LIN {X 0,Y 572.923,Z 346.522,A -85,B 0,C 180,E1 -2106.073,E2 -2106.073} C_VEL
LIN {X 0,Y 572.929,Z 346.988,A -85,B 0,C 180,E1 -2107.123,E2 -2107.123} C_VEL
LIN {X 0,Y 572.933,Z 346.186,A -85,B 0,C 180,E1 -2108.272,E2 -2108.272} C_VEL
LIN {X 0,Y 572.946,Z 344.14,A -85,B 0,C 180,E1 -2109.395,E2 -2109.395} C_VEL
LIN {X 0,Y 573.006,Z 340.639,A -85,B 0,C 180,E1 -2110.546,E2 -2110.546} C_VEL
LIN {X 0,Y 573.022,Z 335.263,A -85,B 0,C 180,E1 -2111.743,E2 -2111.743} C_VEL
LIN {X 0,Y 573.058,Z 329.01,A -85,B 0,C 180,E1 -2112.77,E2 -2112.77} C_VEL
LIN {X 0,Y 573.128,Z 322.073,A -85,B 0,C 180,E1 -2113.656,E2 -2113.656} C_VEL
LIN {X 0,Y 573.173,Z 315.507,A -85,B 0,C 180,E1 -2114.34,E2 -2114.34} C_VEL
LIN {X 0,Y 573.239,Z 307.033,A -85,B 0,C 180,E1 -2115.058,E2 -2115.058} C_VEL
LIN {X 0,Y 573.328,Z 297.887,A -85,B 0,C 180,E1 -2115.675,E2 -2115.675} C_VEL
LIN {X 0,Y 573.423,Z 286.508,A -85,B 0,C 180,E1 -2116.263,E2 -2116.263} C_VEL
LIN {X 0,Y 573.486,Z 274.83,A -85,B 0,C 180,E1 -2116.68,E2 -2116.68} C_VEL
LIN {X 0,Y 573.2,Z 269.025,A -85,B 0,C 180,E1 -2116.842,E2 -2116.842} C_VEL
LIN {X 0,Y 573.003,Z 267.326,A -85,B 0,C 180,E1 -2116.901,E2 -2116.901} C_VEL
LIN {X 0,Y 572.997,Z 260.215,A -85,B 0,C 180,E1 -2119.939,E2 -2119.939} C_VEL
LIN {X 0,Y 572.989,Z 255.042,A -85,B 0,C 180,E1 -2122.173,E2 -2122.173} C_VEL
LIN {X 0,Y 573.027,Z 247.981,A -85,B 0,C 180,E1 -2125.259,E2 -2125.259} C_VEL
LIN {X 0,Y 573.063,Z 241.461,A -85,B 0,C 180,E1 -2128.173,E2 -2128.173} C_VEL
LIN {X 0,Y 573.075,Z 235.778,A -85,B 0,C 180,E1 -2130.623,E2 -2130.623} C_VEL
LIN {X 0,Y 573.068,Z 230.379,A -85,B 0,C 180,E1 -2133.014,E2 -2133.014} C_VEL
LIN {X 0,Y 573.079,Z 224.661,A -85,B 0,C 180,E1 -2135.357,E2 -2135.357} C_VEL
LIN {X 0,Y 573.108,Z 218.041,A -85,B 0,C 180,E1 -2138.036,E2 -2138.036} C_VEL
LIN {X 0,Y 573.12,Z 217.1,A -85,B 0,C 180,E1 -2138.415,E2 -2138.415} C_VEL
LIN {X 0,Y 573.273,Z 217.077,A -85,B 0,C 180,E1 -2140.731,E2 -2140.731} C_VEL
LIN {X 0,Y 573.248,Z 217.082,A -85,B 0,C 180,E1 -2143.621,E2 -2143.621} C_VEL
LIN {X 0,Y 573.231,Z 217.082,A -85,B 0,C 180,E1 -2146.529,E2 -2146.529} C_VEL
LIN {X 0,Y 573.267,Z 217.078,A -85,B 0,C 180,E1 -2148.745,E2 -2148.745} C_VEL
LIN {X 0,Y 573.286,Z 217.076,A -85,B 0,C 180,E1 -2151.54,E2 -2151.54} C_VEL
LIN {X 0,Y 573.284,Z 217.077,A -85,B 0,C 180,E1 -2154.372,E2 -2154.372} C_VEL
LIN {X 0,Y 573.315,Z 217.073,A -85,B 0,C 180,E1 -2157.892,E2 -2157.892} C_VEL
LIN {X 0,Y 573.327,Z 217.07,A -85,B 0,C 180,E1 -2160.702,E2 -2160.702} C_VEL
LIN {X 0,Y 573.307,Z 217.073,A -85,B 0,C 180,E1 -2162.811,E2 -2162.811} C_VEL
LIN {X 0,Y 573.288,Z 217.075,A -85,B 0,C 180,E1 -2165.628,E2 -2165.628} C_VEL
LIN {X 0,Y 573.286,Z 217.078,A -85,B 0,C 180,E1 -2168.459,E2 -2168.459} C_VEL
LIN {X 0,Y 573.276,Z 217.076,A -85,B 0,C 180,E1 -2171.312,E2 -2171.312} C_VEL
LIN {X 0,Y 573.286,Z 217.078,A -85,B 0,C 180,E1 -2174.424,E2 -2174.424} C_VEL
LIN {X 0,Y 573.262,Z 217.079,A -85,B 0,C 180,E1 -2177.111,E2 -2177.111} C_VEL
LIN {X 0,Y 573.246,Z 217.081,A -85,B 0,C 180,E1 -2180.077,E2 -2180.077} C_VEL
LIN {X 0,Y 573.237,Z 217.081,A -85,B 0,C 180,E1 -2182.338,E2 -2182.338} C_VEL
LIN {X 0,Y 573.244,Z 217.081,A -85,B 0,C 180,E1 -2185.411,E2 -2185.411} C_VEL
LIN {X 0,Y 573.239,Z 217.084,A -85,B 0,C 180,E1 -2188.564,E2 -2188.564} C_VEL
LIN {X 0,Y 573.223,Z 217.086,A -85,B 0,C 180,E1 -2190.994,E2 -2190.994} C_VEL
LIN {X 0,Y 573.243,Z 217.083,A -85,B 0,C 180,E1 -2193.521,E2 -2193.521} C_VEL
LIN {X 0,Y 573.218,Z 217.084,A -85,B 0,C 180,E1 -2196.051,E2 -2196.051} C_VEL
LIN {X 0,Y 573.246,Z 217.08,A -85,B 0,C 180,E1 -2198.701,E2 -2198.701} C_VEL
LIN {X 0,Y 573.231,Z 217.084,A -85,B 0,C 180,E1 -2201.593,E2 -2201.593} C_VEL
LIN {X 0,Y 573.236,Z 217.083,A -85,B 0,C 180,E1 -2204.334,E2 -2204.334} C_VEL
LIN {X 0,Y 573.244,Z 217.081,A -85,B 0,C 180,E1 -2207.358,E2 -2207.358} C_VEL
LIN {X 0,Y 573.253,Z 217.079,A -85,B 0,C 180,E1 -2210.568,E2 -2210.568} C_VEL
LIN {X 0,Y 573.279,Z 217.182,A -85,B 0,C 180,E1 -2213.244,E2 -2213.244} C_VEL
LIN {X 0,Y 573.748,Z 221.859,A -85,B 0,C 180,E1 -2214.85,E2 -2214.85} C_VEL
LIN {X 0,Y 573.7,Z 228.345,A -85,B 0,C 180,E1 -2216.966,E2 -2216.966} C_VEL
LIN {X 0,Y 573.556,Z 237.515,A -85,B 0,C 180,E1 -2219.842,E2 -2219.842} C_VEL
LIN {X 0,Y 573.422,Z 246.743,A -85,B 0,C 180,E1 -2222.638,E2 -2222.638} C_VEL
LIN {X 0,Y 573.367,Z 256.185,A -85,B 0,C 180,E1 -2225.37,E2 -2225.37} C_VEL
LIN {X 0,Y 573.349,Z 265.605,A -85,B 0,C 180,E1 -2228.046,E2 -2228.046} C_VEL
LIN {X 0,Y 573.228,Z 276.33,A -85,B 0,C 180,E1 -2231.078,E2 -2231.078} C_VEL
LIN {X 0,Y 573.164,Z 286.788,A -85,B 0,C 180,E1 -2233.985,E2 -2233.985} C_VEL
LIN {X 0,Y 573.094,Z 297.379,A -85,B 0,C 180,E1 -2236.887,E2 -2236.887} C_VEL
LIN {X 0,Y 573.083,Z 299.53,A -85,B 0,C 180,E1 -2237.472,E2 -2237.472} C_VEL
LIN {X 0,Y 573.866,Z 306.371,A -85,B 0,C 180,E1 -2237.624,E2 -2237.624} C_VEL
LIN {X 0,Y 573.779,Z 318.5,A -85,B 0,C 180,E1 -2237.937,E2 -2237.937} C_VEL
LIN {X 0,Y 573.642,Z 330.524,A -85,B 0,C 180,E1 -2238.382,E2 -2238.382} C_VEL
LIN {X 0,Y 573.509,Z 342.485,A -85,B 0,C 180,E1 -2238.977,E2 -2238.977} C_VEL
LIN {X 0,Y 573.446,Z 353.483,A -85,B 0,C 180,E1 -2239.675,E2 -2239.675} C_VEL
LIN {X 0,Y 573.308,Z 363.647,A -85,B 0,C 180,E1 -2240.474,E2 -2240.474} C_VEL
LIN {X 0,Y 573.215,Z 372.787,A -85,B 0,C 180,E1 -2241.362,E2 -2241.362} C_VEL
LIN {X 0,Y 573.142,Z 381.69,A -85,B 0,C 180,E1 -2242.425,E2 -2242.425} C_VEL
LIN {X 0,Y 573.051,Z 388.404,A -85,B 0,C 180,E1 -2243.415,E2 -2243.415} C_VEL
LIN {X 0,Y 573.07,Z 393.68,A -85,B 0,C 180,E1 -2244.37,E2 -2244.37} C_VEL
LIN {X 0,Y 573.028,Z 398.372,A -85,B 0,C 180,E1 -2245.428,E2 -2245.428} C_VEL
LIN {X 0,Y 573.022,Z 401.958,A -85,B 0,C 180,E1 -2246.484,E2 -2246.484} C_VEL
LIN {X 0,Y 572.959,Z 403.808,A -85,B 0,C 180,E1 -2247.188,E2 -2247.188} C_VEL
LIN {X 0,Y 572.94,Z 405.198,A -85,B 0,C 180,E1 -2247.891,E2 -2247.891} C_VEL
LIN {X 0,Y 572.94,Z 406.785,A -85,B 0,C 180,E1 -2249.297,E2 -2249.297} C_VEL
LIN {X 0,Y 572.938,Z 407,A -85,B 0,C 180,E1 -2250,E2 -2250} C_VEL
LIN {X 0,Y 572.946,Z 406.186,A -85,B 0,C 180,E1 -2251.406,E2 -2251.406} C_VEL
LIN {X 0,Y 572.94,Z 405.199,A -85,B 0,C 180,E1 -2252.109,E2 -2252.109} C_VEL
LIN {X 0,Y 572.959,Z 403.81,A -85,B 0,C 180,E1 -2252.812,E2 -2252.812} C_VEL
LIN {X 0,Y 573.015,Z 400.895,A -85,B 0,C 180,E1 -2253.868,E2 -2253.868} C_VEL
LIN {X 0,Y 572.963,Z 396.948,A -85,B 0,C 180,E1 -2254.926,E2 -2254.926} C_VEL
LIN {X 0,Y 573.065,Z 390.876,A -85,B 0,C 180,E1 -2256.16,E2 -2256.16} C_VEL
LIN {X 0,Y 573.119,Z 384.236,A -85,B 0,C 180,E1 -2257.221,E2 -2257.221} C_VEL
LIN {X 0,Y 573.201,Z 375.989,A -85,B 0,C 180,E1 -2258.283,E2 -2258.283} C_VEL
LIN {X 0,Y 573.287,Z 367.537,A -85,B 0,C 180,E1 -2259.17,E2 -2259.17} C_VEL
LIN {X 0,Y 573.425,Z 357.096,A -85,B 0,C 180,E1 -2260.058,E2 -2260.058} C_VEL
LIN {X 0,Y 573.511,Z 345.53,A -85,B 0,C 180,E1 -2260.847,E2 -2260.847} C_VEL
LIN {X 0,Y 573.61,Z 333.88,A -85,B 0,C 180,E1 -2261.466,E2 -2261.466} C_VEL
LIN {X 0,Y 573.758,Z 321.166,A -85,B 0,C 180,E1 -2261.974,E2 -2261.974} C_VEL
LIN {X 0,Y 573.867,Z 308.51,A -85,B 0,C 180,E1 -2262.331,E2 -2262.331} C_VEL
LIN {X 0,Y 573.573,Z 302.638,A -85,B 0,C 180,E1 -2262.455,E2 -2262.455} C_VEL
LIN {X 0,Y 573.084,Z 299.529,A -85,B 0,C 180,E1 -2262.528,E2 -2262.528} C_VEL
LIN {X 0,Y 573.158,Z 289.435,A -85,B 0,C 180,E1 -2265.286,E2 -2265.286} C_VEL
LIN {X 0,Y 573.217,Z 278.843,A -85,B 0,C 180,E1 -2268.219,E2 -2268.219} C_VEL
LIN {X 0,Y 573.3,Z 269.576,A -85,B 0,C 180,E1 -2270.825,E2 -2270.825} C_VEL
LIN {X 0,Y 573.349,Z 260.089,A -85,B 0,C 180,E1 -2273.477,E2 -2273.477} C_VEL
LIN {X 0,Y 573.356,Z 249.227,A -85,B 0,C 180,E1 -2276.516,E2 -2276.516} C_VEL
LIN {X 0,Y 573.441,Z 239.004,A -85,B 0,C 180,E1 -2279.522,E2 -2279.522} C_VEL
LIN {X 0,Y 573.633,Z 230.314,A -85,B 0,C 180,E1 -2282.288,E2 -2282.288} C_VEL
LIN {X 0,Y 573.793,Z 223.076,A -85,B 0,C 180,E1 -2284.851,E2 -2284.851} C_VEL
LIN {X 0,Y 573.73,Z 220.074,A -85,B 0,C 180,E1 -2286.052,E2 -2286.052} C_VEL
LIN {X 0,Y 573.256,Z 217.082,A -85,B 0,C 180,E1 -2287.457,E2 -2287.457} C_VEL
LIN {X 0,Y 573.248,Z 217.083,A -85,B 0,C 180,E1 -2290.525,E2 -2290.525} C_VEL
LIN {X 0,Y 573.242,Z 217.082,A -85,B 0,C 180,E1 -2293.359,E2 -2293.359} C_VEL
LIN {X 0,Y 573.243,Z 217.081,A -85,B 0,C 180,E1 -2296.332,E2 -2296.332} C_VEL
LIN {X 0,Y 573.233,Z 217.082,A -85,B 0,C 180,E1 -2298.543,E2 -2298.543} C_VEL
LIN {X 0,Y 573.247,Z 217.081,A -85,B 0,C 180,E1 -2301.299,E2 -2301.299} C_VEL
LIN {X 0,Y 573.217,Z 217.086,A -85,B 0,C 180,E1 -2304.019,E2 -2304.019} C_VEL
LIN {X 0,Y 573.17,Z 217.102,A -85,B 0,C 180,E1 -2305.665,E2 -2305.665} C_VEL
LIN {X 0,Y 573.151,Z 219.81,A -85,B 0,C 180,E1 -2308.179,E2 -2308.179} C_VEL
LIN {X 0,Y 573.114,Z 222.452,A -85,B 0,C 180,E1 -2310.626,E2 -2310.626} C_VEL
LIN {X 0,Y 573.064,Z 225.599,A -85,B 0,C 180,E1 -2313.543,E2 -2313.543} C_VEL
LIN {X 0,Y 573.028,Z 228.468,A -85,B 0,C 180,E1 -2316.126,E2 -2316.126} C_VEL
LIN {X 0,Y 572.987,Z 231.649,A -85,B 0,C 180,E1 -2319.164,E2 -2319.164} C_VEL
LIN {X 0,Y 572.947,Z 234.241,A -85,B 0,C 180,E1 -2321.402,E2 -2321.402} C_VEL
LIN {X 0,Y 572.957,Z 237.107,A -85,B 0,C 180,E1 -2323.613,E2 -2323.613} C_VEL
LIN {X 0,Y 572.983,Z 240.932,A -85,B 0,C 180,E1 -2326.523,E2 -2326.523} C_VEL
LIN {X 0,Y 572.961,Z 243.669,A -85,B 0,C 180,E1 -2328.581,E2 -2328.581} C_VEL
LIN {X 0,Y 573.844,Z 250.337,A -85,B 0,C 180,E1 -2328.759,E2 -2328.759} C_VEL
LIN {X 0,Y 573.776,Z 263.544,A -85,B 0,C 180,E1 -2329.153,E2 -2329.153} C_VEL
LIN {X 0,Y 573.655,Z 274.091,A -85,B 0,C 180,E1 -2329.589,E2 -2329.589} C_VEL
LIN {X 0,Y 573.527,Z 285.736,A -85,B 0,C 180,E1 -2330.211,E2 -2330.211} C_VEL
LIN {X 0,Y 573.367,Z 297.401,A -85,B 0,C 180,E1 -2331.009,E2 -2331.009} C_VEL
LIN {X 0,Y 573.295,Z 307.756,A -85,B 0,C 180,E1 -2331.896,E2 -2331.896} C_VEL
LIN {X 0,Y 573.167,Z 317.63,A -85,B 0,C 180,E1 -2332.957,E2 -2332.957} C_VEL
LIN {X 0,Y 573.139,Z 325.578,A -85,B 0,C 180,E1 -2334.017,E2 -2334.017} C_VEL
LIN {X 0,Y 573.018,Z 331.94,A -85,B 0,C 180,E1 -2335.075,E2 -2335.075} C_VEL
LIN {X 0,Y 573.04,Z 336.998,A -85,B 0,C 180,E1 -2336.132,E2 -2336.132} C_VEL
LIN {X 0,Y 572.972,Z 340.93,A -85,B 0,C 180,E1 -2337.188,E2 -2337.188} C_VEL
LIN {X 0,Y 572.954,Z 342.953,A -85,B 0,C 180,E1 -2337.891,E2 -2337.891} C_VEL
LIN {X 0,Y 572.949,Z 344.562,A -85,B 0,C 180,E1 -2338.594,E2 -2338.594} C_VEL
LIN {X 0,Y 572.94,Z 345.769,A -85,B 0,C 180,E1 -2339.297,E2 -2339.297} C_VEL
LIN {X 0,Y 572.941,Z 346.555,A -85,B 0,C 180,E1 -2340,E2 -2340} C_VEL
LIN {X 0,Y 572.947,Z 346.926,A -85,B 0,C 180,E1 -2341.406,E2 -2341.406} C_VEL
LIN {X 0,Y 572.938,Z 346.541,A -85,B 0,C 180,E1 -2342.109,E2 -2342.109} C_VEL
LIN {X 0,Y 572.955,Z 345.737,A -85,B 0,C 180,E1 -2342.812,E2 -2342.812} C_VEL
LIN {X 0,Y 573.009,Z 344.519,A -85,B 0,C 180,E1 -2343.516,E2 -2343.516} C_VEL
LIN {X 0,Y 573.005,Z 341.922,A -85,B 0,C 180,E1 -2344.573,E2 -2344.573} C_VEL
LIN {X 0,Y 573.052,Z 338.318,A -85,B 0,C 180,E1 -2345.631,E2 -2345.631} C_VEL
LIN {X 0,Y 573.046,Z 333.102,A -85,B 0,C 180,E1 -2346.788,E2 -2346.788} C_VEL
LIN {X 0,Y 573.112,Z 326.507,A -85,B 0,C 180,E1 -2347.93,E2 -2347.93} C_VEL
LIN {X 0,Y 573.174,Z 318.791,A -85,B 0,C 180,E1 -2348.994,E2 -2348.994} C_VEL
LIN {X 0,Y 573.261,Z 309.1,A -85,B 0,C 180,E1 -2350.061,E2 -2350.061} C_VEL
LIN {X 0,Y 573.399,Z 299.626,A -85,B 0,C 180,E1 -2350.907,E2 -2350.907} C_VEL
LIN {X 0,Y 573.462,Z 289.699,A -85,B 0,C 180,E1 -2351.631,E2 -2351.631} C_VEL
LIN {X 0,Y 573.6,Z 278.331,A -85,B 0,C 180,E1 -2352.292,E2 -2352.292} C_VEL
LIN {X 0,Y 573.745,Z 265.287,A -85,B 0,C 180,E1 -2352.873,E2 -2352.873} C_VEL
LIN {X 0,Y 573.792,Z 252.609,A -85,B 0,C 180,E1 -2353.277,E2 -2353.277} C_VEL
LIN {X 0,Y 573.584,Z 247.706,A -85,B 0,C 180,E1 -2353.4,E2 -2353.4} C_VEL
LIN {X 0,Y 572.987,Z 243.681,A -85,B 0,C 180,E1 -2353.499,E2 -2353.499} C_VEL
LIN {X 0,Y 572.946,Z 239.849,A -85,B 0,C 180,E1 -2356.387,E2 -2356.387} C_VEL
LIN {X 0,Y 572.955,Z 236.331,A -85,B 0,C 180,E1 -2359.073,E2 -2359.073} C_VEL
LIN {X 0,Y 572.307,Z 235.617,A -85,B 0,C 180,E1 -2359.656,E2 -2359.656} C_VEL
LIN {X 0,Y 569.428,Z 234.597,A -85,B 0,C 180,E1 -2360.603,E2 -2360.603} C_VEL
LIN {X 0,Y 566.984,Z 233.82,A -85,B 0,C 180,E1 -2361.365,E2 -2361.365} C_VEL
LIN {X 0,Y 565.94,Z 233.19,A -85,B 0,C 180,E1 -2361.954,E2 -2361.954} C_VEL
LIN {X 0,Y 565.859,Z 232.963,A -85,B 0,C 180,E1 -2362.153,E2 -2362.153} C_VEL
LIN {X 0,Y 565.926,Z 229.746,A -85,B 0,C 180,E1 -2364.976,E2 -2364.976} C_VEL
LIN {X 0,Y 565.956,Z 226.848,A -85,B 0,C 180,E1 -2367.353,E2 -2367.353} C_VEL
LIN {X 0,Y 565.954,Z 223.033,A -85,B 0,C 180,E1 -2370.607,E2 -2370.607} C_VEL
LIN {X 0,Y 565.971,Z 220.055,A -85,B 0,C 180,E1 -2373.119,E2 -2373.119} C_VEL
LIN {X 0,Y 566.033,Z 217.983,A -85,B 0,C 180,E1 -2374.967,E2 -2374.967} C_VEL
LIN {X 0,Y 566.198,Z 217.954,A -85,B 0,C 180,E1 -2377.461,E2 -2377.461} C_VEL
LIN {X 0,Y 566.212,Z 217.957,A -85,B 0,C 180,E1 -2380.199,E2 -2380.199} C_VEL
LIN {X 0,Y 566.201,Z 217.954,A -85,B 0,C 180,E1 -2383.055,E2 -2383.055} C_VEL
LIN {X 0,Y 566.161,Z 217.959,A -85,B 0,C 180,E1 -2386.053,E2 -2386.053} C_VEL
LIN {X 0,Y 566.168,Z 217.96,A -85,B 0,C 180,E1 -2388.859,E2 -2388.859} C_VEL
LIN {X 0,Y 566.185,Z 217.957,A -85,B 0,C 180,E1 -2391.446,E2 -2391.446} C_VEL
LIN {X 0,Y 566.134,Z 217.963,A -85,B 0,C 180,E1 -2394.305,E2 -2394.305} C_VEL
LIN {X 0,Y 566.198,Z 217.956,A -85,B 0,C 180,E1 -2396.896,E2 -2396.896} C_VEL
LIN {X 0,Y 566.172,Z 217.956,A -85,B 0,C 180,E1 -2399.406,E2 -2399.406} C_VEL
LIN {X 0,Y 566.194,Z 217.959,A -85,B 0,C 180,E1 -2401.856,E2 -2401.856} C_VEL
LIN {X 0,Y 566.242,Z 217.948,A -85,B 0,C 180,E1 -2405.039,E2 -2405.039} C_VEL
LIN {X 0,Y 566.199,Z 217.955,A -85,B 0,C 180,E1 -2408.137,E2 -2408.137} C_VEL
LIN {X 0,Y 566.236,Z 217.949,A -85,B 0,C 180,E1 -2410.614,E2 -2410.614} C_VEL
LIN {X 0,Y 566.206,Z 217.957,A -85,B 0,C 180,E1 -2413.412,E2 -2413.412} C_VEL
LIN {X 0,Y 566.183,Z 217.958,A -85,B 0,C 180,E1 -2416.358,E2 -2416.358} C_VEL
LIN {X 0,Y 566.235,Z 217.95,A -85,B 0,C 180,E1 -2419.27,E2 -2419.27} C_VEL
LIN {X 0,Y 566.193,Z 217.96,A -85,B 0,C 180,E1 -2422.152,E2 -2422.152} C_VEL
LIN {X 0,Y 566.249,Z 217.946,A -85,B 0,C 180,E1 -2425.016,E2 -2425.016} C_VEL
LIN {X 0,Y 566.281,Z 217.951,A -85,B 0,C 180,E1 -2427.866,E2 -2427.866} C_VEL
LIN {X 0,Y 566.291,Z 217.945,A -85,B 0,C 180,E1 -2430,E2 -2430} C_VEL
LIN {X 0,Y 566.262,Z 217.946,A -85,B 0,C 180,E1 -2432.846,E2 -2432.846} C_VEL
LIN {X 0,Y 566.104,Z 217.974,A -85,B 0,C 180,E1 -2435.432,E2 -2435.432} C_VEL
LIN {X 0,Y 566.069,Z 223.635,A -85,B 0,C 180,E1 -2437.849,E2 -2437.849} C_VEL
LIN {X 0,Y 566.02,Z 230.292,A -85,B 0,C 180,E1 -2440.734,E2 -2440.734} C_VEL
LIN {X 0,Y 566.033,Z 236.901,A -85,B 0,C 180,E1 -2443.645,E2 -2443.645} C_VEL
LIN {X 0,Y 566.018,Z 243.637,A -85,B 0,C 180,E1 -2446.594,E2 -2446.594} C_VEL
LIN {X 0,Y 565.952,Z 250.222,A -85,B 0,C 180,E1 -2449.59,E2 -2449.59} C_VEL
LIN {X 0,Y 565.909,Z 255.385,A -85,B 0,C 180,E1 -2451.874,E2 -2451.874} C_VEL
LIN {X 0,Y 565.923,Z 262.492,A -85,B 0,C 180,E1 -2454.976,E2 -2454.976} C_VEL
LIN {X 0,Y 565.904,Z 267.364,A -85,B 0,C 180,E1 -2457.08,E2 -2457.08} C_VEL
LIN {X 0,Y 566.513,Z 274.523,A -85,B 0,C 180,E1 -2457.282,E2 -2457.282} C_VEL
LIN {X 0,Y 566.417,Z 285.729,A -85,B 0,C 180,E1 -2457.679,E2 -2457.679} C_VEL
LIN {X 0,Y 566.322,Z 296.517,A -85,B 0,C 180,E1 -2458.224,E2 -2458.224} C_VEL
LIN {X 0,Y 566.216,Z 305.993,A -85,B 0,C 180,E1 -2458.852,E2 -2458.852} C_VEL
LIN {X 0,Y 566.136,Z 313.899,A -85,B 0,C 180,E1 -2459.508,E2 -2459.508} C_VEL
LIN {X 0,Y 566.08,Z 320.632,A -85,B 0,C 180,E1 -2460.187,E2 -2460.187} C_VEL
LIN {X 0,Y 565.994,Z 327.532,A -85,B 0,C 180,E1 -2461.043,E2 -2461.043} C_VEL
LIN {X 0,Y 565.959,Z 332.829,A -85,B 0,C 180,E1 -2461.854,E2 -2461.854} C_VEL
LIN {X 0,Y 565.909,Z 337.404,A -85,B 0,C 180,E1 -2462.727,E2 -2462.727} C_VEL
LIN {X 0,Y 565.923,Z 341.287,A -85,B 0,C 180,E1 -2463.69,E2 -2463.69} C_VEL
LIN {X 0,Y 565.865,Z 344.555,A -85,B 0,C 180,E1 -2464.842,E2 -2464.842} C_VEL
LIN {X 0,Y 565.823,Z 346.612,A -85,B 0,C 180,E1 -2466.161,E2 -2466.161} C_VEL
LIN {X 0,Y 565.811,Z 346.826,A -85,B 0,C 180,E1 -2467.491,E2 -2467.491} C_VEL
LIN {X 0,Y 565.827,Z 345.878,A -85,B 0,C 180,E1 -2468.509,E2 -2468.509} C_VEL
LIN {X 0,Y 565.874,Z 343.601,A -85,B 0,C 180,E1 -2469.644,E2 -2469.644} C_VEL
LIN {X 0,Y 565.934,Z 340.054,A -85,B 0,C 180,E1 -2470.753,E2 -2470.753} C_VEL
LIN {X 0,Y 565.941,Z 335.107,A -85,B 0,C 180,E1 -2471.832,E2 -2471.832} C_VEL
LIN {X 0,Y 565.969,Z 329.973,A -85,B 0,C 180,E1 -2472.7,E2 -2472.7} C_VEL
LIN {X 0,Y 566.065,Z 323.648,A -85,B 0,C 180,E1 -2473.556,E2 -2473.556} C_VEL
LIN {X 0,Y 566.121,Z 315.656,A -85,B 0,C 180,E1 -2474.416,E2 -2474.416} C_VEL
LIN {X 0,Y 566.2,Z 307.008,A -85,B 0,C 180,E1 -2475.159,E2 -2475.159} C_VEL
LIN {X 0,Y 566.298,Z 297.369,A -85,B 0,C 180,E1 -2475.815,E2 -2475.815} C_VEL
LIN {X 0,Y 566.44,Z 285.522,A -85,B 0,C 180,E1 -2476.419,E2 -2476.419} C_VEL
LIN {X 0,Y 566.501,Z 274.585,A -85,B 0,C 180,E1 -2476.806,E2 -2476.806} C_VEL
LIN {X 0,Y 565.911,Z 267.362,A -85,B 0,C 180,E1 -2477.01,E2 -2477.01} C_VEL
LIN {X 0,Y 565.915,Z 260.969,A -85,B 0,C 180,E1 -2479.776,E2 -2479.776} C_VEL
LIN {X 0,Y 565.916,Z 254.427,A -85,B 0,C 180,E1 -2482.637,E2 -2482.637} C_VEL
LIN {X 0,Y 565.97,Z 248.805,A -85,B 0,C 180,E1 -2485.165,E2 -2485.165} C_VEL
LIN {X 0,Y 565.995,Z 243.137,A -85,B 0,C 180,E1 -2487.728,E2 -2487.728} C_VEL
LIN {X 0,Y 566.008,Z 237.008,A -85,B 0,C 180,E1 -2490.363,E2 -2490.363} C_VEL
LIN {X 0,Y 566.005,Z 230.057,A -85,B 0,C 180,E1 -2493.382,E2 -2493.382} C_VEL
LIN {X 0,Y 565.989,Z 224.225,A -85,B 0,C 180,E1 -2495.81,E2 -2495.81} C_VEL
LIN {X 0,Y 566.051,Z 217.98,A -85,B 0,C 180,E1 -2498.337,E2 -2498.337} C_VEL
LIN {X 0,Y 566.234,Z 217.954,A -85,B 0,C 180,E1 -2500.614,E2 -2500.614} C_VEL
LIN {X 0,Y 566.214,Z 217.959,A -85,B 0,C 180,E1 -2503.412,E2 -2503.412} C_VEL
LIN {X 0,Y 566.194,Z 217.959,A -85,B 0,C 180,E1 -2506.359,E2 -2506.359} C_VEL
LIN {X 0,Y 566.239,Z 217.953,A -85,B 0,C 180,E1 -2508.675,E2 -2508.675} C_VEL
LIN {X 0,Y 566.23,Z 217.955,A -85,B 0,C 180,E1 -2511.434,E2 -2511.434} C_VEL
LIN {X 0,Y 566.252,Z 217.953,A -85,B 0,C 180,E1 -2514.302,E2 -2514.302} C_VEL
LIN {X 0,Y 566.286,Z 217.949,A -85,B 0,C 180,E1 -2517.866,E2 -2517.866} C_VEL
LIN {X 0,Y 566.299,Z 217.945,A -85,B 0,C 180,E1 -2520.711,E2 -2520.711} C_VEL
LIN {X 0,Y 566.273,Z 217.949,A -85,B 0,C 180,E1 -2522.845,E2 -2522.845} C_VEL
LIN {X 0,Y 566.256,Z 217.951,A -85,B 0,C 180,E1 -2525.698,E2 -2525.698} C_VEL
LIN {X 0,Y 566.23,Z 217.956,A -85,B 0,C 180,E1 -2528.566,E2 -2528.566} C_VEL
LIN {X 0,Y 566.246,Z 217.952,A -85,B 0,C 180,E1 -2531.454,E2 -2531.454} C_VEL
LIN {X 0,Y 566.239,Z 217.955,A -85,B 0,C 180,E1 -2534.507,E2 -2534.507} C_VEL
LIN {X 0,Y 566.202,Z 217.957,A -85,B 0,C 180,E1 -2537.332,E2 -2537.332} C_VEL
LIN {X 0,Y 566.211,Z 217.96,A -85,B 0,C 180,E1 -2540.337,E2 -2540.337} C_VEL
LIN {X 0,Y 566.175,Z 217.961,A -85,B 0,C 180,E1 -2543.281,E2 -2543.281} C_VEL
LIN {X 0,Y 566.209,Z 217.957,A -85,B 0,C 180,E1 -2545.749,E2 -2545.749} C_VEL
LIN {X 0,Y 566.206,Z 217.957,A -85,B 0,C 180,E1 -2548.202,E2 -2548.202} C_VEL
LIN {X 0,Y 566.189,Z 217.962,A -85,B 0,C 180,E1 -2551.076,E2 -2551.076} C_VEL
LIN {X 0,Y 566.2,Z 217.958,A -85,B 0,C 180,E1 -2553.732,E2 -2553.732} C_VEL
LIN {X 0,Y 566.203,Z 217.957,A -85,B 0,C 180,E1 -2556.57,E2 -2556.57} C_VEL
LIN {X 0,Y 566.218,Z 217.956,A -85,B 0,C 180,E1 -2559.686,E2 -2559.686} C_VEL
LIN {X 0,Y 566.204,Z 217.961,A -85,B 0,C 180,E1 -2562.917,E2 -2562.917} C_VEL
LIN {X 0,Y 566.197,Z 217.959,A -85,B 0,C 180,E1 -2566.049,E2 -2566.049} C_VEL
LIN {X 0,Y 566.206,Z 217.957,A -85,B 0,C 180,E1 -2569.215,E2 -2569.215} C_VEL
LIN {X 0,Y 566.188,Z 217.961,A -85,B 0,C 180,E1 -2571.637,E2 -2571.637} C_VEL
LIN {X 0,Y 566.237,Z 217.996,A -85,B 0,C 180,E1 -2572.989,E2 -2572.989} C_VEL
LIN {X 0,Y 566.779,Z 221.851,A -85,B 0,C 180,E1 -2574.353,E2 -2574.353} C_VEL
LIN {X 0,Y 566.734,Z 229.603,A -85,B 0,C 180,E1 -2576.932,E2 -2576.932} C_VEL
LIN {X 0,Y 566.615,Z 237.454,A -85,B 0,C 180,E1 -2579.433,E2 -2579.433} C_VEL
LIN {X 0,Y 566.427,Z 246.649,A -85,B 0,C 180,E1 -2582.271,E2 -2582.271} C_VEL
LIN {X 0,Y 566.354,Z 256.072,A -85,B 0,C 180,E1 -2585.045,E2 -2585.045} C_VEL
LIN {X 0,Y 566.296,Z 265.475,A -85,B 0,C 180,E1 -2587.758,E2 -2587.758} C_VEL
LIN {X 0,Y 566.207,Z 275.583,A -85,B 0,C 180,E1 -2590.621,E2 -2590.621} C_VEL
LIN {X 0,Y 566.126,Z 285.464,A -85,B 0,C 180,E1 -2593.41,E2 -2593.41} C_VEL
LIN {X 0,Y 566.045,Z 296.055,A -85,B 0,C 180,E1 -2596.355,E2 -2596.355} C_VEL
LIN {X 0,Y 566.012,Z 299.53,A -85,B 0,C 180,E1 -2597.313,E2 -2597.313} C_VEL
LIN {X 0,Y 566.932,Z 306.37,A -85,B 0,C 180,E1 -2597.471,E2 -2597.471} C_VEL
LIN {X 0,Y 566.84,Z 318.501,A -85,B 0,C 180,E1 -2597.787,E2 -2597.787} C_VEL
LIN {X 0,Y 566.68,Z 330.316,A -85,B 0,C 180,E1 -2598.228,E2 -2598.228} C_VEL
LIN {X 0,Y 566.532,Z 342.984,A -85,B 0,C 180,E1 -2598.868,E2 -2598.868} C_VEL
LIN {X 0,Y 566.434,Z 354.746,A -85,B 0,C 180,E1 -2599.636,E2 -2599.636} C_VEL
LIN {X 0,Y 566.301,Z 363.647,A -85,B 0,C 180,E1 -2600.355,E2 -2600.355} C_VEL
LIN {X 0,Y 566.166,Z 372.787,A -85,B 0,C 180,E1 -2601.254,E2 -2601.254} C_VEL
LIN {X 0,Y 566.08,Z 381.69,A -85,B 0,C 180,E1 -2602.33,E2 -2602.33} C_VEL
LIN {X 0,Y 565.967,Z 388.956,A -85,B 0,C 180,E1 -2603.422,E2 -2603.422} C_VEL
LIN {X 0,Y 566.004,Z 393.68,A -85,B 0,C 180,E1 -2604.299,E2 -2604.299} C_VEL
LIN {X 0,Y 565.933,Z 398.373,A -85,B 0,C 180,E1 -2605.37,E2 -2605.37} C_VEL
LIN {X 0,Y 565.927,Z 401.958,A -85,B 0,C 180,E1 -2606.44,E2 -2606.44} C_VEL
LIN {X 0,Y 565.878,Z 403.808,A -85,B 0,C 180,E1 -2607.153,E2 -2607.153} C_VEL
LIN {X 0,Y 565.846,Z 406.185,A -85,B 0,C 180,E1 -2608.577,E2 -2608.577} C_VEL
LIN {X 0,Y 565.839,Z 407,A -85,B 0,C 180,E1 -2610,E2 -2610} C_VEL
LIN {X 0,Y 565.846,Z 406.186,A -85,B 0,C 180,E1 -2611.424,E2 -2611.424} C_VEL
LIN {X 0,Y 565.878,Z 403.81,A -85,B 0,C 180,E1 -2612.848,E2 -2612.848} C_VEL
LIN {X 0,Y 565.926,Z 400.895,A -85,B 0,C 180,E1 -2613.917,E2 -2613.917} C_VEL
LIN {X 0,Y 565.878,Z 396.948,A -85,B 0,C 180,E1 -2614.988,E2 -2614.988} C_VEL
LIN {X 0,Y 566.002,Z 391.866,A -85,B 0,C 180,E1 -2616.059,E2 -2616.059} C_VEL
LIN {X 0,Y 566.04,Z 385.467,A -85,B 0,C 180,E1 -2617.132,E2 -2617.132} C_VEL
LIN {X 0,Y 566.134,Z 377.477,A -85,B 0,C 180,E1 -2618.208,E2 -2618.208} C_VEL
LIN {X 0,Y 566.229,Z 369.333,A -85,B 0,C 180,E1 -2619.106,E2 -2619.106} C_VEL
LIN {X 0,Y 566.344,Z 359.398,A -85,B 0,C 180,E1 -2620.005,E2 -2620.005} C_VEL
LIN {X 0,Y 566.501,Z 348.331,A -85,B 0,C 180,E1 -2620.805,E2 -2620.805} C_VEL
LIN {X 0,Y 566.609,Z 335.942,A -85,B 0,C 180,E1 -2621.51,E2 -2621.51} C_VEL
LIN {X 0,Y 566.748,Z 323.762,A -85,B 0,C 180,E1 -2622.034,E2 -2622.034} C_VEL
LIN {X 0,Y 566.927,Z 310.339,A -85,B 0,C 180,E1 -2622.439,E2 -2622.439} C_VEL
LIN {X 0,Y 566.64,Z 303.505,A -85,B 0,C 180,E1 -2622.593,E2 -2622.593} C_VEL
LIN {X 0,Y 566.012,Z 299.529,A -85,B 0,C 180,E1 -2622.687,E2 -2622.687} C_VEL
LIN {X 0,Y 566.089,Z 289.435,A -85,B 0,C 180,E1 -2625.481,E2 -2625.481} C_VEL
LIN {X 0,Y 566.176,Z 278.843,A -85,B 0,C 180,E1 -2628.454,E2 -2628.454} C_VEL
LIN {X 0,Y 566.24,Z 269.401,A -85,B 0,C 180,E1 -2631.097,E2 -2631.097} C_VEL
LIN {X 0,Y 566.291,Z 259.78,A -85,B 0,C 180,E1 -2633.788,E2 -2633.788} C_VEL
LIN {X 0,Y 566.313,Z 249.59,A -85,B 0,C 180,E1 -2636.68,E2 -2636.68} C_VEL
LIN {X 0,Y 566.433,Z 239.523,A -85,B 0,C 180,E1 -2639.712,E2 -2639.712} C_VEL
LIN {X 0,Y 566.652,Z 230.995,A -85,B 0,C 180,E1 -2642.501,E2 -2642.501} C_VEL
LIN {X 0,Y 566.849,Z 224.743,A -85,B 0,C 180,E1 -2644.773,E2 -2644.773} C_VEL
LIN {X 0,Y 566.714,Z 221.072,A -85,B 0,C 180,E1 -2646.284,E2 -2646.284} C_VEL
LIN {X 0,Y 566.214,Z 217.959,A -85,B 0,C 180,E1 -2647.797,E2 -2647.797} C_VEL
LIN {X 0,Y 566.207,Z 217.959,A -85,B 0,C 180,E1 -2650.786,E2 -2650.786} C_VEL
LIN {X 0,Y 566.202,Z 217.96,A -85,B 0,C 180,E1 -2653.951,E2 -2653.951} C_VEL
LIN {X 0,Y 566.205,Z 217.958,A -85,B 0,C 180,E1 -2657.083,E2 -2657.083} C_VEL
LIN {X 0,Y 566.219,Z 217.958,A -85,B 0,C 180,E1 -2660.314,E2 -2660.314} C_VEL
LIN {X 0,Y 566.204,Z 217.959,A -85,B 0,C 180,E1 -2663.43,E2 -2663.43} C_VEL
LIN {X 0,Y 566.179,Z 217.963,A -85,B 0,C 180,E1 -2665.18,E2 -2665.18} C_VEL
LIN {X 0,Y 566.142,Z 218.667,A -85,B 0,C 180,E1 -2666.277,E2 -2666.277} C_VEL
LIN {X 0,Y 566.093,Z 221.454,A -85,B 0,C 180,E1 -2668.941,E2 -2668.941} C_VEL
LIN {X 0,Y 566.043,Z 224.542,A -85,B 0,C 180,E1 -2671.848,E2 -2671.848} C_VEL
LIN {X 0,Y 566.04,Z 227.908,A -85,B 0,C 180,E1 -2675.01,E2 -2675.01} C_VEL
LIN {X 0,Y 565.926,Z 230.469,A -85,B 0,C 180,E1 -2677.358,E2 -2677.358} C_VEL
LIN {X 0,Y 565.898,Z 232.875,A -85,B 0,C 180,E1 -2679.651,E2 -2679.651} C_VEL
LIN {X 0,Y 565.856,Z 235.335,A -85,B 0,C 180,E1 -2681.91,E2 -2681.91} C_VEL
LIN {X 0,Y 565.848,Z 238.082,A -85,B 0,C 180,E1 -2684.142,E2 -2684.142} C_VEL
LIN {X 0,Y 565.882,Z 240.95,A -85,B 0,C 180,E1 -2686.351,E2 -2686.351} C_VEL
LIN {X 0,Y 565.899,Z 243.882,A -85,B 0,C 180,E1 -2688.443,E2 -2688.443} C_VEL
LIN {X 0,Y 566.883,Z 251.23,A -85,B 0,C 180,E1 -2688.627,E2 -2688.627} C_VEL
LIN {X 0,Y 566.834,Z 262.781,A -85,B 0,C 180,E1 -2688.979,E2 -2688.979} C_VEL
LIN {X 0,Y 566.698,Z 274.382,A -85,B 0,C 180,E1 -2689.46,E2 -2689.46} C_VEL
LIN {X 0,Y 566.525,Z 285.944,A -85,B 0,C 180,E1 -2690.089,E2 -2690.089} C_VEL
LIN {X 0,Y 566.367,Z 297.574,A -85,B 0,C 180,E1 -2690.897,E2 -2690.897} C_VEL
LIN {X 0,Y 566.263,Z 307.891,A -85,B 0,C 180,E1 -2691.794,E2 -2691.794} C_VEL
LIN {X 0,Y 566.12,Z 317.739,A -85,B 0,C 180,E1 -2692.869,E2 -2692.869} C_VEL
LIN {X 0,Y 566.084,Z 325.667,A -85,B 0,C 180,E1 -2693.942,E2 -2693.942} C_VEL
LIN {X 0,Y 565.928,Z 332.007,A -85,B 0,C 180,E1 -2695.013,E2 -2695.013} C_VEL
LIN {X 0,Y 565.947,Z 337.051,A -85,B 0,C 180,E1 -2696.084,E2 -2696.084} C_VEL
LIN {X 0,Y 565.892,Z 340.969,A -85,B 0,C 180,E1 -2697.153,E2 -2697.153} C_VEL
LIN {X 0,Y 565.858,Z 342.986,A -85,B 0,C 180,E1 -2697.865,E2 -2697.865} C_VEL
LIN {X 0,Y 565.849,Z 344.589,A -85,B 0,C 180,E1 -2698.577,E2 -2698.577} C_VEL
LIN {X 0,Y 565.841,Z 345.79,A -85,B 0,C 180,E1 -2699.288,E2 -2699.288} C_VEL
LIN {X 0,Y 565.841,Z 346.563,A -85,B 0,C 180,E1 -2700,E2 -2700} C_VEL
LIN {X 0,Y 565.846,Z 346.922,A -85,B 0,C 180,E1 -2701.424,E2 -2701.424} C_VEL
LIN {X 0,Y 565.839,Z 346.531,A -85,B 0,C 180,E1 -2702.136,E2 -2702.136} C_VEL
LIN {X 0,Y 565.874,Z 345.717,A -85,B 0,C 180,E1 -2702.848,E2 -2702.848} C_VEL
LIN {X 0,Y 565.915,Z 344.493,A -85,B 0,C 180,E1 -2703.56,E2 -2703.56} C_VEL
LIN {X 0,Y 565.896,Z 341.883,A -85,B 0,C 180,E1 -2704.63,E2 -2704.63} C_VEL
LIN {X 0,Y 565.978,Z 338.266,A -85,B 0,C 180,E1 -2705.701,E2 -2705.701} C_VEL
LIN {X 0,Y 565.972,Z 332.719,A -85,B 0,C 180,E1 -2706.936,E2 -2706.936} C_VEL
LIN {X 0,Y 566.04,Z 326.425,A -85,B 0,C 180,E1 -2708.029,E2 -2708.029} C_VEL
LIN {X 0,Y 566.127,Z 318.681,A -85,B 0,C 180,E1 -2709.107,E2 -2709.107} C_VEL
LIN {X 0,Y 566.244,Z 308.967,A -85,B 0,C 180,E1 -2710.187,E2 -2710.187} C_VEL
LIN {X 0,Y 566.392,Z 299.87,A -85,B 0,C 180,E1 -2711.009,E2 -2711.009} C_VEL
LIN {X 0,Y 566.447,Z 288.926,A -85,B 0,C 180,E1 -2711.813,E2 -2711.813} C_VEL
LIN {X 0,Y 566.63,Z 278.071,A -85,B 0,C 180,E1 -2712.445,E2 -2712.445} C_VEL
LIN {X 0,Y 566.792,Z 266.086,A -85,B 0,C 180,E1 -2712.988,E2 -2712.988} C_VEL
LIN {X 0,Y 566.861,Z 252.986,A -85,B 0,C 180,E1 -2713.42,E2 -2713.42} C_VEL
LIN {X 0,Y 566.52,Z 247.595,A -85,B 0,C 180,E1 -2713.559,E2 -2713.559} C_VEL
LIN {X 0,Y 565.895,Z 243.663,A -85,B 0,C 180,E1 -2713.672,E2 -2713.672} C_VEL
LIN {X 0,Y 565.856,Z 239.83,A -85,B 0,C 180,E1 -2716.599,E2 -2716.599} C_VEL
LIN {X 0,Y 565.85,Z 235.967,A -85,B 0,C 180,E1 -2719.594,E2 -2719.594} C_VEL
LIN {X 0,Y 565.859,Z 232.963,A -85,B 0,C 180,E1 -2722.153,E2 -2722.153} C_VEL
LIN {X 0,Y 565.2,Z 232.337,A -85,B 0,C 180,E1 -2722.744,E2 -2722.744} C_VEL
LIN {X 0,Y 562.342,Z 231.465,A -85,B 0,C 180,E1 -2723.704,E2 -2723.704} C_VEL
LIN {X 0,Y 559.935,Z 230.788,A -85,B 0,C 180,E1 -2724.477,E2 -2724.477} C_VEL
LIN {X 0,Y 558.919,Z 230.128,A -85,B 0,C 180,E1 -2725.072,E2 -2725.072} C_VEL
LIN {X 0,Y 558.846,Z 229.883,A -85,B 0,C 180,E1 -2725.273,E2 -2725.273} C_VEL
LIN {X 0,Y 558.867,Z 226.927,A -85,B 0,C 180,E1 -2727.729,E2 -2727.729} C_VEL
LIN {X 0,Y 558.912,Z 223.139,A -85,B 0,C 180,E1 -2731.035,E2 -2731.035} C_VEL
LIN {X 0,Y 558.938,Z 219.749,A -85,B 0,C 180,E1 -2733.914,E2 -2733.914} C_VEL
LIN {X 0,Y 558.941,Z 219.122,A -85,B 0,C 180,E1 -2734.46,E2 -2734.46} C_VEL
LIN {X 0,Y 559.103,Z 218.844,A -85,B 0,C 180,E1 -2736.439,E2 -2736.439} C_VEL
LIN {X 0,Y 559.18,Z 218.828,A -85,B 0,C 180,E1 -2738.934,E2 -2738.934} C_VEL
LIN {X 0,Y 559.165,Z 218.837,A -85,B 0,C 180,E1 -2741.77,E2 -2741.77} C_VEL
LIN {X 0,Y 559.136,Z 218.833,A -85,B 0,C 180,E1 -2744.74,E2 -2744.74} C_VEL
LIN {X 0,Y 559.143,Z 218.833,A -85,B 0,C 180,E1 -2747.867,E2 -2747.867} C_VEL
LIN {X 0,Y 559.177,Z 218.827,A -85,B 0,C 180,E1 -2750.134,E2 -2750.134} C_VEL
LIN {X 0,Y 559.114,Z 218.843,A -85,B 0,C 180,E1 -2752.889,E2 -2752.889} C_VEL
LIN {X 0,Y 559.155,Z 218.832,A -85,B 0,C 180,E1 -2756.053,E2 -2756.053} C_VEL
LIN {X 0,Y 559.153,Z 218.832,A -85,B 0,C 180,E1 -2758.98,E2 -2758.98} C_VEL
LIN {X 0,Y 559.149,Z 218.834,A -85,B 0,C 180,E1 -2761.623,E2 -2761.623} C_VEL
LIN {X 0,Y 559.168,Z 218.836,A -85,B 0,C 180,E1 -2763.902,E2 -2763.902} C_VEL
LIN {X 0,Y 559.144,Z 218.832,A -85,B 0,C 180,E1 -2766.572,E2 -2766.572} C_VEL
LIN {X 0,Y 559.181,Z 218.834,A -85,B 0,C 180,E1 -2769.395,E2 -2769.395} C_VEL
LIN {X 0,Y 559.139,Z 218.836,A -85,B 0,C 180,E1 -2771.685,E2 -2771.685} C_VEL
LIN {X 0,Y 559.16,Z 218.83,A -85,B 0,C 180,E1 -2773.947,E2 -2773.947} C_VEL
LIN {X 0,Y 559.159,Z 218.831,A -85,B 0,C 180,E1 -2776.184,E2 -2776.184} C_VEL
LIN {X 0,Y 559.194,Z 218.828,A -85,B 0,C 180,E1 -2779.133,E2 -2779.133} C_VEL
LIN {X 0,Y 559.146,Z 218.836,A -85,B 0,C 180,E1 -2782.053,E2 -2782.053} C_VEL
LIN {X 0,Y 559.225,Z 218.822,A -85,B 0,C 180,E1 -2784.953,E2 -2784.953} C_VEL
LIN {X 0,Y 559.251,Z 218.827,A -85,B 0,C 180,E1 -2787.839,E2 -2787.839} C_VEL
LIN {X 0,Y 559.26,Z 218.821,A -85,B 0,C 180,E1 -2790,E2 -2790} C_VEL
LIN {X 0,Y 559.231,Z 218.823,A -85,B 0,C 180,E1 -2792.881,E2 -2792.881} C_VEL
LIN {X 0,Y 559.061,Z 218.851,A -85,B 0,C 180,E1 -2795.41,E2 -2795.41} C_VEL
LIN {X 0,Y 559.016,Z 224.601,A -85,B 0,C 180,E1 -2797.949,E2 -2797.949} C_VEL
LIN {X 0,Y 559.015,Z 232.309,A -85,B 0,C 180,E1 -2801.295,E2 -2801.295} C_VEL
LIN {X 0,Y 558.963,Z 239.691,A -85,B 0,C 180,E1 -2804.564,E2 -2804.564} C_VEL
LIN {X 0,Y 558.934,Z 246.39,A -85,B 0,C 180,E1 -2807.564,E2 -2807.564} C_VEL
LIN {X 0,Y 558.852,Z 251.372,A -85,B 0,C 180,E1 -2809.849,E2 -2809.849} C_VEL
LIN {X 0,Y 558.823,Z 256.523,A -85,B 0,C 180,E1 -2812.166,E2 -2812.166} C_VEL
LIN {X 0,Y 558.815,Z 263.144,A -85,B 0,C 180,E1 -2815.106,E2 -2815.106} C_VEL
LIN {X 0,Y 558.812,Z 267.349,A -85,B 0,C 180,E1 -2816.946,E2 -2816.946} C_VEL
LIN {X 0,Y 559.533,Z 274.583,A -85,B 0,C 180,E1 -2817.161,E2 -2817.161} C_VEL
LIN {X 0,Y 559.42,Z 285.365,A -85,B 0,C 180,E1 -2817.547,E2 -2817.547} C_VEL
LIN {X 0,Y 559.294,Z 296.555,A -85,B 0,C 180,E1 -2818.114,E2 -2818.114} C_VEL
LIN {X 0,Y 559.17,Z 305.814,A -85,B 0,C 180,E1 -2818.734,E2 -2818.734} C_VEL
LIN {X 0,Y 559.104,Z 313.304,A -85,B 0,C 180,E1 -2819.356,E2 -2819.356} C_VEL
LIN {X 0,Y 559.046,Z 319.587,A -85,B 0,C 180,E1 -2819.98,E2 -2819.98} C_VEL
LIN {X 0,Y 558.943,Z 326.507,A -85,B 0,C 180,E1 -2820.823,E2 -2820.823} C_VEL
LIN {X 0,Y 558.907,Z 332.33,A -85,B 0,C 180,E1 -2821.703,E2 -2821.703} C_VEL
LIN {X 0,Y 558.822,Z 336.984,A -85,B 0,C 180,E1 -2822.581,E2 -2822.581} C_VEL
LIN {X 0,Y 558.826,Z 341.112,A -85,B 0,C 180,E1 -2823.598,E2 -2823.598} C_VEL
LIN {X 0,Y 558.793,Z 343.73,A -85,B 0,C 180,E1 -2824.47,E2 -2824.47} C_VEL
LIN {X 0,Y 558.751,Z 345.573,A -85,B 0,C 180,E1 -2825.352,E2 -2825.352} C_VEL
LIN {X 0,Y 558.734,Z 346.726,A -85,B 0,C 180,E1 -2826.387,E2 -2826.387} C_VEL
LIN {X 0,Y 558.717,Z 346.982,A -85,B 0,C 180,E1 -2827.141,E2 -2827.141} C_VEL
LIN {X 0,Y 558.724,Z 346.515,A -85,B 0,C 180,E1 -2828.051,E2 -2828.051} C_VEL
LIN {X 0,Y 558.745,Z 345.221,A -85,B 0,C 180,E1 -2828.97,E2 -2828.97} C_VEL
LIN {X 0,Y 558.806,Z 343.05,A -85,B 0,C 180,E1 -2829.898,E2 -2829.898} C_VEL
LIN {X 0,Y 558.829,Z 339.199,A -85,B 0,C 180,E1 -2831.011,E2 -2831.011} C_VEL
LIN {X 0,Y 558.865,Z 333.963,A -85,B 0,C 180,E1 -2832.101,E2 -2832.101} C_VEL
LIN {X 0,Y 558.917,Z 328.604,A -85,B 0,C 180,E1 -2832.97,E2 -2832.97} C_VEL
LIN {X 0,Y 558.975,Z 322.683,A -85,B 0,C 180,E1 -2833.75,E2 -2833.75} C_VEL
LIN {X 0,Y 559.05,Z 316.179,A -85,B 0,C 180,E1 -2834.458,E2 -2834.458} C_VEL
LIN {X 0,Y 559.151,Z 307.995,A -85,B 0,C 180,E1 -2835.183,E2 -2835.183} C_VEL
LIN {X 0,Y 559.27,Z 299.204,A -85,B 0,C 180,E1 -2835.808,E2 -2835.808} C_VEL
LIN {X 0,Y 559.35,Z 290.775,A -85,B 0,C 180,E1 -2836.286,E2 -2836.286} C_VEL
LIN {X 0,Y 559.461,Z 282.155,A -85,B 0,C 180,E1 -2836.669,E2 -2836.669} C_VEL
LIN {X 0,Y 559.514,Z 273.369,A -85,B 0,C 180,E1 -2836.964,E2 -2836.964} C_VEL
LIN {X 0,Y 558.817,Z 267.327,A -85,B 0,C 180,E1 -2837.154,E2 -2837.154} C_VEL
LIN {X 0,Y 558.837,Z 260.594,A -85,B 0,C 180,E1 -2840.105,E2 -2840.105} C_VEL
LIN {X 0,Y 558.826,Z 254.461,A -85,B 0,C 180,E1 -2842.867,E2 -2842.867} C_VEL
LIN {X 0,Y 558.917,Z 247.557,A -85,B 0,C 180,E1 -2846.089,E2 -2846.089} C_VEL
LIN {X 0,Y 558.926,Z 240.9,A -85,B 0,C 180,E1 -2848.966,E2 -2848.966} C_VEL
LIN {X 0,Y 558.945,Z 234.728,A -85,B 0,C 180,E1 -2851.662,E2 -2851.662} C_VEL
LIN {X 0,Y 558.972,Z 227.181,A -85,B 0,C 180,E1 -2854.859,E2 -2854.859} C_VEL
LIN {X 0,Y 558.966,Z 219.847,A -85,B 0,C 180,E1 -2857.84,E2 -2857.84} C_VEL
LIN {X 0,Y 559.017,Z 218.856,A -85,B 0,C 180,E1 -2858.29,E2 -2858.29} C_VEL
LIN {X 0,Y 559.196,Z 218.83,A -85,B 0,C 180,E1 -2860.494,E2 -2860.494} C_VEL
LIN {X 0,Y 559.183,Z 218.833,A -85,B 0,C 180,E1 -2863.197,E2 -2863.197} C_VEL
LIN {X 0,Y 559.168,Z 218.834,A -85,B 0,C 180,E1 -2866.184,E2 -2866.184} C_VEL
LIN {X 0,Y 559.199,Z 218.831,A -85,B 0,C 180,E1 -2869.133,E2 -2869.133} C_VEL
LIN {X 0,Y 559.208,Z 218.83,A -85,B 0,C 180,E1 -2872.054,E2 -2872.054} C_VEL
LIN {X 0,Y 559.254,Z 218.823,A -85,B 0,C 180,E1 -2874.953,E2 -2874.953} C_VEL
LIN {X 0,Y 559.257,Z 218.825,A -85,B 0,C 180,E1 -2877.839,E2 -2877.839} C_VEL
LIN {X 0,Y 559.27,Z 218.821,A -85,B 0,C 180,E1 -2880.72,E2 -2880.72} C_VEL
LIN {X 0,Y 559.24,Z 218.825,A -85,B 0,C 180,E1 -2882.881,E2 -2882.881} C_VEL
LIN {X 0,Y 559.224,Z 218.827,A -85,B 0,C 180,E1 -2885.77,E2 -2885.77} C_VEL
LIN {X 0,Y 559.188,Z 218.832,A -85,B 0,C 180,E1 -2888.674,E2 -2888.674} C_VEL
LIN {X 0,Y 559.209,Z 218.828,A -85,B 0,C 180,E1 -2891.6,E2 -2891.6} C_VEL
LIN {X 0,Y 559.204,Z 218.831,A -85,B 0,C 180,E1 -2894.595,E2 -2894.595} C_VEL
LIN {X 0,Y 559.145,Z 218.837,A -85,B 0,C 180,E1 -2897.557,E2 -2897.557} C_VEL
LIN {X 0,Y 559.169,Z 218.833,A -85,B 0,C 180,E1 -2899.837,E2 -2899.837} C_VEL
LIN {X 0,Y 559.143,Z 218.836,A -85,B 0,C 180,E1 -2902.153,E2 -2902.153} C_VEL
LIN {X 0,Y 559.146,Z 218.839,A -85,B 0,C 180,E1 -2905.179,E2 -2905.179} C_VEL
LIN {X 0,Y 559.144,Z 218.838,A -85,B 0,C 180,E1 -2907.714,E2 -2907.714} C_VEL
LIN {X 0,Y 559.151,Z 218.836,A -85,B 0,C 180,E1 -2910.183,E2 -2910.183} C_VEL
LIN {X 0,Y 559.155,Z 218.835,A -85,B 0,C 180,E1 -2912.715,E2 -2912.715} C_VEL
LIN {X 0,Y 559.131,Z 218.838,A -85,B 0,C 180,E1 -2915.324,E2 -2915.324} C_VEL
LIN {X 0,Y 559.136,Z 218.839,A -85,B 0,C 180,E1 -2918.017,E2 -2918.017} C_VEL
LIN {X 0,Y 559.158,Z 218.836,A -85,B 0,C 180,E1 -2920.812,E2 -2920.812} C_VEL
LIN {X 0,Y 559.143,Z 218.837,A -85,B 0,C 180,E1 -2923.734,E2 -2923.734} C_VEL
LIN {X 0,Y 559.148,Z 218.837,A -85,B 0,C 180,E1 -2926.804,E2 -2926.804} C_VEL
LIN {X 0,Y 559.158,Z 218.835,A -85,B 0,C 180,E1 -2929.188,E2 -2929.188} C_VEL
LIN {X 0,Y 559.135,Z 218.84,A -85,B 0,C 180,E1 -2931.982,E2 -2931.982} C_VEL
LIN {X 0,Y 559.215,Z 219.002,A -85,B 0,C 180,E1 -2932.799,E2 -2932.799} C_VEL
LIN {X 0,Y 559.82,Z 224.299,A -85,B 0,C 180,E1 -2934.688,E2 -2934.688} C_VEL
LIN {X 0,Y 559.758,Z 230.863,A -85,B 0,C 180,E1 -2936.896,E2 -2936.896} C_VEL
LIN {X 0,Y 559.622,Z 238.702,A -85,B 0,C 180,E1 -2939.428,E2 -2939.428} C_VEL
LIN {X 0,Y 559.423,Z 247.923,A -85,B 0,C 180,E1 -2942.301,E2 -2942.301} C_VEL
LIN {X 0,Y 559.314,Z 257.412,A -85,B 0,C 180,E1 -2945.14,E2 -2945.14} C_VEL
LIN {X 0,Y 559.245,Z 266.63,A -85,B 0,C 180,E1 -2947.851,E2 -2947.851} C_VEL
LIN {X 0,Y 559.145,Z 275.921,A -85,B 0,C 180,E1 -2950.509,E2 -2950.509} C_VEL
LIN {X 0,Y 559.074,Z 285.464,A -85,B 0,C 180,E1 -2953.194,E2 -2953.194} C_VEL
LIN {X 0,Y 558.994,Z 296.055,A -85,B 0,C 180,E1 -2956.18,E2 -2956.18} C_VEL
LIN {X 0,Y 558.937,Z 299.53,A -85,B 0,C 180,E1 -2957.15,E2 -2957.15} C_VEL
LIN {X 0,Y 560.018,Z 307.51,A -85,B 0,C 180,E1 -2957.336,E2 -2957.336} C_VEL
LIN {X 0,Y 559.9,Z 319.875,A -85,B 0,C 180,E1 -2957.679,E2 -2957.679} C_VEL
LIN {X 0,Y 559.718,Z 332.281,A -85,B 0,C 180,E1 -2958.171,E2 -2958.171} C_VEL
LIN {X 0,Y 559.555,Z 343.773,A -85,B 0,C 180,E1 -2958.773,E2 -2958.773} C_VEL
LIN {X 0,Y 559.424,Z 354.745,A -85,B 0,C 180,E1 -2959.504,E2 -2959.504} C_VEL
LIN {X 0,Y 559.244,Z 365.6,A -85,B 0,C 180,E1 -2960.415,E2 -2960.415} C_VEL
LIN {X 0,Y 559.127,Z 374.413,A -85,B 0,C 180,E1 -2961.325,E2 -2961.325} C_VEL
LIN {X 0,Y 558.996,Z 383.003,A -85,B 0,C 180,E1 -2962.414,E2 -2962.414} C_VEL
LIN {X 0,Y 558.884,Z 390.687,A -85,B 0,C 180,E1 -2963.649,E2 -2963.649} C_VEL
LIN {X 0,Y 558.869,Z 395.366,A -85,B 0,C 180,E1 -2964.588,E2 -2964.588} C_VEL
LIN {X 0,Y 558.868,Z 399.677,A -85,B 0,C 180,E1 -2965.673,E2 -2965.673} C_VEL
LIN {X 0,Y 558.836,Z 401.958,A -85,B 0,C 180,E1 -2966.395,E2 -2966.395} C_VEL
LIN {X 0,Y 558.799,Z 403.808,A -85,B 0,C 180,E1 -2967.116,E2 -2967.116} C_VEL
LIN {X 0,Y 558.745,Z 406.184,A -85,B 0,C 180,E1 -2968.559,E2 -2968.559} C_VEL
LIN {X 0,Y 558.74,Z 407,A -85,B 0,C 180,E1 -2970,E2 -2970} C_VEL
LIN {X 0,Y 558.745,Z 406.185,A -85,B 0,C 180,E1 -2971.442,E2 -2971.442} C_VEL
LIN {X 0,Y 558.799,Z 403.81,A -85,B 0,C 180,E1 -2972.884,E2 -2972.884} C_VEL
LIN {X 0,Y 558.844,Z 400.895,A -85,B 0,C 180,E1 -2973.966,E2 -2973.966} C_VEL
LIN {X 0,Y 558.798,Z 396.948,A -85,B 0,C 180,E1 -2975.051,E2 -2975.051} C_VEL
LIN {X 0,Y 558.922,Z 391.866,A -85,B 0,C 180,E1 -2976.136,E2 -2976.136} C_VEL
LIN {X 0,Y 558.977,Z 385.466,A -85,B 0,C 180,E1 -2977.223,E2 -2977.223} C_VEL
LIN {X 0,Y 559.099,Z 377.476,A -85,B 0,C 180,E1 -2978.312,E2 -2978.312} C_VEL
LIN {X 0,Y 559.195,Z 369.333,A -85,B 0,C 180,E1 -2979.221,E2 -2979.221} C_VEL
LIN {X 0,Y 559.358,Z 359.397,A -85,B 0,C 180,E1 -2980.131,E2 -2980.131} C_VEL
LIN {X 0,Y 559.511,Z 348.441,A -85,B 0,C 180,E1 -2980.935,E2 -2980.935} C_VEL
LIN {X 0,Y 559.636,Z 336.813,A -85,B 0,C 180,E1 -2981.61,E2 -2981.61} C_VEL
LIN {X 0,Y 559.794,Z 324.975,A -85,B 0,C 180,E1 -2982.139,E2 -2982.139} C_VEL
LIN {X 0,Y 559.99,Z 312.167,A -85,B 0,C 180,E1 -2982.549,E2 -2982.549} C_VEL
LIN {X 0,Y 559.815,Z 304.929,A -85,B 0,C 180,E1 -2982.72,E2 -2982.72} C_VEL
LIN {X 0,Y 558.938,Z 299.529,A -85,B 0,C 180,E1 -2982.85,E2 -2982.85} C_VEL
LIN {X 0,Y 559.054,Z 289.435,A -85,B 0,C 180,E1 -2985.681,E2 -2985.681} C_VEL
LIN {X 0,Y 559.143,Z 278.751,A -85,B 0,C 180,E1 -2988.694,E2 -2988.694} C_VEL
LIN {X 0,Y 559.171,Z 268.374,A -85,B 0,C 180,E1 -2991.553,E2 -2991.553} C_VEL
LIN {X 0,Y 559.229,Z 258.014,A -85,B 0,C 180,E1 -2994.502,E2 -2994.502} C_VEL
LIN {X 0,Y 559.283,Z 249.786,A -85,B 0,C 180,E1 -2996.897,E2 -2996.897} C_VEL
LIN {X 0,Y 559.419,Z 240.053,A -85,B 0,C 180,E1 -2999.905,E2 -2999.905} C_VEL
LIN {X 0,Y 559.678,Z 231.68,A -85,B 0,C 180,E1 -3002.718,E2 -3002.718} C_VEL
LIN {X 0,Y 559.889,Z 226.044,A -85,B 0,C 180,E1 -3004.83,E2 -3004.83} C_VEL
LIN {X 0,Y 559.718,Z 222.087,A -85,B 0,C 180,E1 -3006.524,E2 -3006.524} C_VEL
LIN {X 0,Y 559.146,Z 218.839,A -85,B 0,C 180,E1 -3008.246,E2 -3008.246} C_VEL
LIN {X 0,Y 559.164,Z 218.835,A -85,B 0,C 180,E1 -3011.051,E2 -3011.051} C_VEL
LIN {X 0,Y 559.145,Z 218.838,A -85,B 0,C 180,E1 -3013.734,E2 -3013.734} C_VEL
LIN {X 0,Y 559.149,Z 218.839,A -85,B 0,C 180,E1 -3016.804,E2 -3016.804} C_VEL
LIN {X 0,Y 559.16,Z 218.838,A -85,B 0,C 180,E1 -3019.188,E2 -3019.188} C_VEL
LIN {X 0,Y 559.138,Z 218.84,A -85,B 0,C 180,E1 -3021.983,E2 -3021.983} C_VEL
LIN {X 0,Y 559.127,Z 218.841,A -85,B 0,C 180,E1 -3024.789,E2 -3024.789} C_VEL
LIN {X 0,Y 559.104,Z 218.876,A -85,B 0,C 180,E1 -3025.552,E2 -3025.552} C_VEL
LIN {X 0,Y 559.058,Z 222.105,A -85,B 0,C 180,E1 -3028.743,E2 -3028.743} C_VEL
LIN {X 0,Y 559.01,Z 225.126,A -85,B 0,C 180,E1 -3031.65,E2 -3031.65} C_VEL
LIN {X 0,Y 558.973,Z 228.488,A -85,B 0,C 180,E1 -3034.859,E2 -3034.859} C_VEL
LIN {X 0,Y 558.876,Z 231.684,A -85,B 0,C 180,E1 -3037.836,E2 -3037.836} C_VEL
LIN {X 0,Y 558.825,Z 234.92,A -85,B 0,C 180,E1 -3040.914,E2 -3040.914} C_VEL
LIN {X 0,Y 558.813,Z 237.407,A -85,B 0,C 180,E1 -3043.186,E2 -3043.186} C_VEL
LIN {X 0,Y 558.782,Z 240.969,A -85,B 0,C 180,E1 -3046.174,E2 -3046.174} C_VEL
LIN {X 0,Y 558.791,Z 243.678,A -85,B 0,C 180,E1 -3048.267,E2 -3048.267} C_VEL
LIN {X 0,Y 559.961,Z 252.025,A -85,B 0,C 180,E1 -3048.492,E2 -3048.492} C_VEL
LIN {X 0,Y 559.888,Z 263.791,A -85,B 0,C 180,E1 -3048.863,E2 -3048.863} C_VEL
LIN {X 0,Y 559.743,Z 274.671,A -85,B 0,C 180,E1 -3049.327,E2 -3049.327} C_VEL
LIN {X 0,Y 559.534,Z 286.153,A -85,B 0,C 180,E1 -3049.963,E2 -3049.963} C_VEL
LIN {X 0,Y 559.375,Z 297.745,A -85,B 0,C 180,E1 -3050.782,E2 -3050.782} C_VEL
LIN {X 0,Y 559.232,Z 308.023,A -85,B 0,C 180,E1 -3051.69,E2 -3051.69} C_VEL
LIN {X 0,Y 559.062,Z 317.849,A -85,B 0,C 180,E1 -3052.778,E2 -3052.778} C_VEL
LIN {X 0,Y 559.03,Z 325.755,A -85,B 0,C 180,E1 -3053.866,E2 -3053.866} C_VEL
LIN {X 0,Y 558.84,Z 332.074,A -85,B 0,C 180,E1 -3054.95,E2 -3054.95} C_VEL
LIN {X 0,Y 558.862,Z 337.103,A -85,B 0,C 180,E1 -3056.034,E2 -3056.034} C_VEL
LIN {X 0,Y 558.815,Z 341.008,A -85,B 0,C 180,E1 -3057.117,E2 -3057.117} C_VEL
LIN {X 0,Y 558.766,Z 343.018,A -85,B 0,C 180,E1 -3057.838,E2 -3057.838} C_VEL
LIN {X 0,Y 558.749,Z 344.616,A -85,B 0,C 180,E1 -3058.559,E2 -3058.559} C_VEL
LIN {X 0,Y 558.741,Z 345.81,A -85,B 0,C 180,E1 -3059.279,E2 -3059.279} C_VEL
LIN {X 0,Y 558.742,Z 346.571,A -85,B 0,C 180,E1 -3060,E2 -3060} C_VEL
LIN {X 0,Y 558.746,Z 346.919,A -85,B 0,C 180,E1 -3061.442,E2 -3061.442} C_VEL
LIN {X 0,Y 558.745,Z 346.521,A -85,B 0,C 180,E1 -3062.163,E2 -3062.163} C_VEL
LIN {X 0,Y 558.796,Z 345.697,A -85,B 0,C 180,E1 -3062.884,E2 -3062.884} C_VEL
LIN {X 0,Y 558.825,Z 344.465,A -85,B 0,C 180,E1 -3063.605,E2 -3063.605} C_VEL
LIN {X 0,Y 558.792,Z 341.844,A -85,B 0,C 180,E1 -3064.689,E2 -3064.689} C_VEL
LIN {X 0,Y 558.876,Z 337.164,A -85,B 0,C 180,E1 -3066.041,E2 -3066.041} C_VEL
LIN {X 0,Y 558.904,Z 331.64,A -85,B 0,C 180,E1 -3067.224,E2 -3067.224} C_VEL
LIN {X 0,Y 558.994,Z 325.157,A -85,B 0,C 180,E1 -3068.313,E2 -3068.313} C_VEL
LIN {X 0,Y 559.07,Z 317.081,A -85,B 0,C 180,E1 -3069.406,E2 -3069.406} C_VEL
LIN {X 0,Y 559.228,Z 308.835,A -85,B 0,C 180,E1 -3070.317,E2 -3070.317} C_VEL
LIN {X 0,Y 559.362,Z 298.932,A -85,B 0,C 180,E1 -3071.215,E2 -3071.215} C_VEL
LIN {X 0,Y 559.47,Z 288.719,A -85,B 0,C 180,E1 -3071.963,E2 -3071.963} C_VEL
LIN {X 0,Y 559.677,Z 277.809,A -85,B 0,C 180,E1 -3072.602,E2 -3072.602} C_VEL
LIN {X 0,Y 559.833,Z 265.749,A -85,B 0,C 180,E1 -3073.152,E2 -3073.152} C_VEL
LIN {X 0,Y 559.926,Z 253.351,A -85,B 0,C 180,E1 -3073.566,E2 -3073.566} C_VEL
LIN {X 0,Y 559.551,Z 248.273,A -85,B 0,C 180,E1 -3073.702,E2 -3073.702} C_VEL
LIN {X 0,Y 558.801,Z 243.675,A -85,B 0,C 180,E1 -3073.825,E2 -3073.825} C_VEL
LIN {X 0,Y 558.772,Z 239.475,A -85,B 0,C 180,E1 -3077.078,E2 -3077.078} C_VEL
LIN {X 0,Y 558.777,Z 236.166,A -85,B 0,C 180,E1 -3079.852,E2 -3079.852} C_VEL
LIN {X 0,Y 558.791,Z 233.486,A -85,B 0,C 180,E1 -3082.168,E2 -3082.168} C_VEL
LIN {X 0,Y 558.828,Z 230.807,A -85,B 0,C 180,E1 -3084.521,E2 -3084.521} C_VEL
LIN {X 0,Y 558.846,Z 229.883,A -85,B 0,C 180,E1 -3085.273,E2 -3085.273} C_VEL
LIN {X 0,Y 558.208,Z 229.205,A -85,B 0,C 180,E1 -3085.871,E2 -3085.871} C_VEL
LIN {X 0,Y 555.365,Z 228.26,A -85,B 0,C 180,E1 -3086.844,E2 -3086.844} C_VEL
LIN {X 0,Y 552.938,Z 227.535,A -85,B 0,C 180,E1 -3087.627,E2 -3087.627} C_VEL
LIN {X 0,Y 551.883,Z 226.927,A -85,B 0,C 180,E1 -3088.231,E2 -3088.231} C_VEL
LIN {X 0,Y 551.791,Z 226.702,A -85,B 0,C 180,E1 -3088.435,E2 -3088.435} C_VEL
LIN {X 0,Y 551.832,Z 223.204,A -85,B 0,C 180,E1 -3091.478,E2 -3091.478} C_VEL
LIN {X 0,Y 551.868,Z 220.132,A -85,B 0,C 180,E1 -3094.129,E2 -3094.129} C_VEL
LIN {X 0,Y 552.03,Z 219.726,A -85,B 0,C 180,E1 -3095.848,E2 -3095.848} C_VEL
LIN {X 0,Y 552.123,Z 219.709,A -85,B 0,C 180,E1 -3098.589,E2 -3098.589} C_VEL
LIN {X 0,Y 552.124,Z 219.71,A -85,B 0,C 180,E1 -3101.446,E2 -3101.446} C_VEL
LIN {X 0,Y 552.093,Z 219.71,A -85,B 0,C 180,E1 -3104.531,E2 -3104.531} C_VEL
LIN {X 0,Y 552.111,Z 219.713,A -85,B 0,C 180,E1 -3107.587,E2 -3107.587} C_VEL
LIN {X 0,Y 552.103,Z 219.71,A -85,B 0,C 180,E1 -3110.47,E2 -3110.47} C_VEL
LIN {X 0,Y 552.053,Z 219.717,A -85,B 0,C 180,E1 -3113.325,E2 -3113.325} C_VEL
LIN {X 0,Y 552.099,Z 219.71,A -85,B 0,C 180,E1 -3115.937,E2 -3115.937} C_VEL
LIN {X 0,Y 552.124,Z 219.712,A -85,B 0,C 180,E1 -3118.541,E2 -3118.541} C_VEL
LIN {X 0,Y 552.106,Z 219.709,A -85,B 0,C 180,E1 -3121.442,E2 -3121.442} C_VEL
LIN {X 0,Y 552.127,Z 219.709,A -85,B 0,C 180,E1 -3124.355,E2 -3124.355} C_VEL
LIN {X 0,Y 552.101,Z 219.71,A -85,B 0,C 180,E1 -3126.758,E2 -3126.758} C_VEL
LIN {X 0,Y 552.124,Z 219.711,A -85,B 0,C 180,E1 -3129.12,E2 -3129.12} C_VEL
LIN {X 0,Y 552.12,Z 219.713,A -85,B 0,C 180,E1 -3131.444,E2 -3131.444} C_VEL
LIN {X 0,Y 552.109,Z 219.71,A -85,B 0,C 180,E1 -3133.737,E2 -3133.737} C_VEL
LIN {X 0,Y 552.123,Z 219.707,A -85,B 0,C 180,E1 -3136.004,E2 -3136.004} C_VEL
LIN {X 0,Y 552.163,Z 219.705,A -85,B 0,C 180,E1 -3138.993,E2 -3138.993} C_VEL
LIN {X 0,Y 552.114,Z 219.711,A -85,B 0,C 180,E1 -3141.951,E2 -3141.951} C_VEL
LIN {X 0,Y 552.203,Z 219.697,A -85,B 0,C 180,E1 -3144.889,E2 -3144.889} C_VEL
LIN {X 0,Y 552.222,Z 219.702,A -85,B 0,C 180,E1 -3147.812,E2 -3147.812} C_VEL
LIN {X 0,Y 552.229,Z 219.697,A -85,B 0,C 180,E1 -3150,E2 -3150} C_VEL
LIN {X 0,Y 552.199,Z 219.699,A -85,B 0,C 180,E1 -3152.918,E2 -3152.918} C_VEL
LIN {X 0,Y 551.981,Z 219.733,A -85,B 0,C 180,E1 -3155.525,E2 -3155.525} C_VEL
LIN {X 0,Y 551.947,Z 225.568,A -85,B 0,C 180,E1 -3158.051,E2 -3158.051} C_VEL
LIN {X 0,Y 551.959,Z 233.057,A -85,B 0,C 180,E1 -3161.353,E2 -3161.353} C_VEL
LIN {X 0,Y 551.916,Z 240.408,A -85,B 0,C 180,E1 -3164.585,E2 -3164.585} C_VEL
LIN {X 0,Y 551.894,Z 246.328,A -85,B 0,C 180,E1 -3167.238,E2 -3167.238} C_VEL
LIN {X 0,Y 551.772,Z 252.523,A -85,B 0,C 180,E1 -3170.115,E2 -3170.115} C_VEL
LIN {X 0,Y 551.748,Z 257.852,A -85,B 0,C 180,E1 -3172.466,E2 -3172.466} C_VEL
LIN {X 0,Y 551.731,Z 263.869,A -85,B 0,C 180,E1 -3175.256,E2 -3175.256} C_VEL
LIN {X 0,Y 551.738,Z 267.436,A -85,B 0,C 180,E1 -3176.828,E2 -3176.828} C_VEL
LIN {X 0,Y 552.53,Z 275.393,A -85,B 0,C 180,E1 -3177.058,E2 -3177.058} C_VEL
LIN {X 0,Y 552.385,Z 287.468,A -85,B 0,C 180,E1 -3177.517,E2 -3177.517} C_VEL
LIN {X 0,Y 552.242,Z 297.994,A -85,B 0,C 180,E1 -3178.091,E2 -3178.091} C_VEL
LIN {X 0,Y 552.127,Z 306.884,A -85,B 0,C 180,E1 -3178.715,E2 -3178.715} C_VEL
LIN {X 0,Y 552.046,Z 314.239,A -85,B 0,C 180,E1 -3179.35,E2 -3179.35} C_VEL
LIN {X 0,Y 551.973,Z 320.723,A -85,B 0,C 180,E1 -3180.024,E2 -3180.024} C_VEL
LIN {X 0,Y 551.868,Z 327.052,A -85,B 0,C 180,E1 -3180.822,E2 -3180.822} C_VEL
LIN {X 0,Y 551.84,Z 332.642,A -85,B 0,C 180,E1 -3181.691,E2 -3181.691} C_VEL
LIN {X 0,Y 551.753,Z 336.166,A -85,B 0,C 180,E1 -3182.343,E2 -3182.343} C_VEL
LIN {X 0,Y 551.713,Z 339.948,A -85,B 0,C 180,E1 -3183.213,E2 -3183.213} C_VEL
LIN {X 0,Y 551.717,Z 342.913,A -85,B 0,C 180,E1 -3184.106,E2 -3184.106} C_VEL
LIN {X 0,Y 551.671,Z 344.988,A -85,B 0,C 180,E1 -3184.979,E2 -3184.979} C_VEL
LIN {X 0,Y 551.639,Z 346.333,A -85,B 0,C 180,E1 -3185.877,E2 -3185.877} C_VEL
LIN {X 0,Y 551.641,Z 346.912,A -85,B 0,C 180,E1 -3186.783,E2 -3186.783} C_VEL
LIN {X 0,Y 551.621,Z 346.672,A -85,B 0,C 180,E1 -3187.822,E2 -3187.822} C_VEL
LIN {X 0,Y 551.654,Z 345.21,A -85,B 0,C 180,E1 -3189.001,E2 -3189.001} C_VEL
LIN {X 0,Y 551.706,Z 342.394,A -85,B 0,C 180,E1 -3190.153,E2 -3190.153} C_VEL
LIN {X 0,Y 551.74,Z 339.88,A -85,B 0,C 180,E1 -3190.895,E2 -3190.895} C_VEL
LIN {X 0,Y 551.781,Z 335.286,A -85,B 0,C 180,E1 -3191.924,E2 -3191.924} C_VEL
LIN {X 0,Y 551.836,Z 329.262,A -85,B 0,C 180,E1 -3192.95,E2 -3192.95} C_VEL
LIN {X 0,Y 551.907,Z 322.803,A -85,B 0,C 180,E1 -3193.821,E2 -3193.821} C_VEL
LIN {X 0,Y 552.002,Z 316.49,A -85,B 0,C 180,E1 -3194.521,E2 -3194.521} C_VEL
LIN {X 0,Y 552.101,Z 308.916,A -85,B 0,C 180,E1 -3195.213,E2 -3195.213} C_VEL
LIN {X 0,Y 552.247,Z 300.802,A -85,B 0,C 180,E1 -3195.815,E2 -3195.815} C_VEL
LIN {X 0,Y 552.327,Z 292.691,A -85,B 0,C 180,E1 -3196.304,E2 -3196.304} C_VEL
LIN {X 0,Y 552.428,Z 283.645,A -85,B 0,C 180,E1 -3196.733,E2 -3196.733} C_VEL
LIN {X 0,Y 552.511,Z 274.132,A -85,B 0,C 180,E1 -3197.068,E2 -3197.068} C_VEL
LIN {X 0,Y 551.721,Z 267.321,A -85,B 0,C 180,E1 -3197.287,E2 -3197.287} C_VEL
LIN {X 0,Y 551.776,Z 260.406,A -85,B 0,C 180,E1 -3200.442,E2 -3200.442} C_VEL
LIN {X 0,Y 551.787,Z 254.052,A -85,B 0,C 180,E1 -3203.362,E2 -3203.362} C_VEL
LIN {X 0,Y 551.856,Z 247.522,A -85,B 0,C 180,E1 -3206.359,E2 -3206.359} C_VEL
LIN {X 0,Y 551.856,Z 240.63,A -85,B 0,C 180,E1 -3209.375,E2 -3209.375} C_VEL
LIN {X 0,Y 551.874,Z 234.84,A -85,B 0,C 180,E1 -3211.888,E2 -3211.888} C_VEL
LIN {X 0,Y 551.903,Z 228.197,A -85,B 0,C 180,E1 -3214.706,E2 -3214.706} C_VEL
LIN {X 0,Y 551.905,Z 220.32,A -85,B 0,C 180,E1 -3217.935,E2 -3217.935} C_VEL
LIN {X 0,Y 551.945,Z 219.738,A -85,B 0,C 180,E1 -3218.232,E2 -3218.232} C_VEL
LIN {X 0,Y 552.154,Z 219.708,A -85,B 0,C 180,E1 -3220.674,E2 -3220.674} C_VEL
LIN {X 0,Y 552.115,Z 219.713,A -85,B 0,C 180,E1 -3223.737,E2 -3223.737} C_VEL
LIN {X 0,Y 552.134,Z 219.712,A -85,B 0,C 180,E1 -3226.004,E2 -3226.004} C_VEL
LIN {X 0,Y 552.167,Z 219.707,A -85,B 0,C 180,E1 -3228.993,E2 -3228.993} C_VEL
LIN {X 0,Y 552.161,Z 219.708,A -85,B 0,C 180,E1 -3231.951,E2 -3231.951} C_VEL
LIN {X 0,Y 552.228,Z 219.698,A -85,B 0,C 180,E1 -3234.889,E2 -3234.889} C_VEL
LIN {X 0,Y 552.228,Z 219.701,A -85,B 0,C 180,E1 -3237.812,E2 -3237.812} C_VEL
LIN {X 0,Y 552.241,Z 219.697,A -85,B 0,C 180,E1 -3240.729,E2 -3240.729} C_VEL
LIN {X 0,Y 552.206,Z 219.701,A -85,B 0,C 180,E1 -3242.918,E2 -3242.918} C_VEL
LIN {X 0,Y 552.194,Z 219.704,A -85,B 0,C 180,E1 -3245.844,E2 -3245.844} C_VEL
LIN {X 0,Y 552.156,Z 219.707,A -85,B 0,C 180,E1 -3248.786,E2 -3248.786} C_VEL
LIN {X 0,Y 552.166,Z 219.707,A -85,B 0,C 180,E1 -3251.75,E2 -3251.75} C_VEL
LIN {X 0,Y 552.14,Z 219.71,A -85,B 0,C 180,E1 -3254.748,E2 -3254.748} C_VEL
LIN {X 0,Y 552.102,Z 219.716,A -85,B 0,C 180,E1 -3257.789,E2 -3257.789} C_VEL
LIN {X 0,Y 552.13,Z 219.712,A -85,B 0,C 180,E1 -3260.101,E2 -3260.101} C_VEL
LIN {X 0,Y 552.095,Z 219.716,A -85,B 0,C 180,E1 -3262.451,E2 -3262.451} C_VEL
LIN {X 0,Y 552.111,Z 219.714,A -85,B 0,C 180,E1 -3265.34,E2 -3265.34} C_VEL
LIN {X 0,Y 552.105,Z 219.713,A -85,B 0,C 180,E1 -3268.099,E2 -3268.099} C_VEL
LIN {X 0,Y 552.101,Z 219.714,A -85,B 0,C 180,E1 -3270.609,E2 -3270.609} C_VEL
LIN {X 0,Y 552.11,Z 219.714,A -85,B 0,C 180,E1 -3273.186,E2 -3273.186} C_VEL
LIN {X 0,Y 552.089,Z 219.718,A -85,B 0,C 180,E1 -3275.844,E2 -3275.844} C_VEL
LIN {X 0,Y 552.12,Z 219.712,A -85,B 0,C 180,E1 -3278.589,E2 -3278.589} C_VEL
LIN {X 0,Y 552.123,Z 219.712,A -85,B 0,C 180,E1 -3281.446,E2 -3281.446} C_VEL
LIN {X 0,Y 552.095,Z 219.715,A -85,B 0,C 180,E1 -3284.532,E2 -3284.532} C_VEL
LIN {X 0,Y 552.132,Z 219.713,A -85,B 0,C 180,E1 -3287.585,E2 -3287.585} C_VEL
LIN {X 0,Y 552.135,Z 219.71,A -85,B 0,C 180,E1 -3290.473,E2 -3290.473} C_VEL
LIN {X 0,Y 552.171,Z 219.905,A -85,B 0,C 180,E1 -3292.572,E2 -3292.572} C_VEL
LIN {X 0,Y 552.889,Z 225.036,A -85,B 0,C 180,E1 -3294.442,E2 -3294.442} C_VEL
LIN {X 0,Y 552.796,Z 232.12,A -85,B 0,C 180,E1 -3296.86,E2 -3296.86} C_VEL
LIN {X 0,Y 552.627,Z 239.943,A -85,B 0,C 180,E1 -3299.423,E2 -3299.423} C_VEL
LIN {X 0,Y 552.397,Z 249.138,A -85,B 0,C 180,E1 -3302.33,E2 -3302.33} C_VEL
LIN {X 0,Y 552.27,Z 258.454,A -85,B 0,C 180,E1 -3305.169,E2 -3305.169} C_VEL
LIN {X 0,Y 552.184,Z 267.786,A -85,B 0,C 180,E1 -3307.947,E2 -3307.947} C_VEL
LIN {X 0,Y 552.071,Z 277.153,A -85,B 0,C 180,E1 -3310.671,E2 -3310.671} C_VEL
LIN {X 0,Y 551.995,Z 286.697,A -85,B 0,C 180,E1 -3313.353,E2 -3313.353} C_VEL
LIN {X 0,Y 551.916,Z 297.379,A -85,B 0,C 180,E1 -3316.374,E2 -3316.374} C_VEL
LIN {X 0,Y 551.886,Z 299.53,A -85,B 0,C 180,E1 -3316.983,E2 -3316.983} C_VEL
LIN {X 0,Y 553.099,Z 308.521,A -85,B 0,C 180,E1 -3317.199,E2 -3317.199} C_VEL
LIN {X 0,Y 552.942,Z 321.175,A -85,B 0,C 180,E1 -3317.568,E2 -3317.568} C_VEL
LIN {X 0,Y 552.743,Z 333.491,A -85,B 0,C 180,E1 -3318.076,E2 -3318.076} C_VEL
LIN {X 0,Y 552.576,Z 345.23,A -85,B 0,C 180,E1 -3318.717,E2 -3318.717} C_VEL
LIN {X 0,Y 552.423,Z 357.094,A -85,B 0,C 180,E1 -3319.555,E2 -3319.555} C_VEL
LIN {X 0,Y 552.201,Z 367.54,A -85,B 0,C 180,E1 -3320.476,E2 -3320.476} C_VEL
LIN {X 0,Y 552.082,Z 375.992,A -85,B 0,C 180,E1 -3321.398,E2 -3321.398} C_VEL
LIN {X 0,Y 551.926,Z 384.236,A -85,B 0,C 180,E1 -3322.5,E2 -3322.5} C_VEL
LIN {X 0,Y 551.821,Z 391.207,A -85,B 0,C 180,E1 -3323.662,E2 -3323.662} C_VEL
LIN {X 0,Y 551.723,Z 396.95,A -85,B 0,C 180,E1 -3324.884,E2 -3324.884} C_VEL
LIN {X 0,Y 551.764,Z 400.895,A -85,B 0,C 180,E1 -3325.983,E2 -3325.983} C_VEL
LIN {X 0,Y 551.723,Z 403.807,A -85,B 0,C 180,E1 -3327.079,E2 -3327.079} C_VEL
LIN {X 0,Y 551.645,Z 406.184,A -85,B 0,C 180,E1 -3328.54,E2 -3328.54} C_VEL
LIN {X 0,Y 551.64,Z 407,A -85,B 0,C 180,E1 -3330,E2 -3330} C_VEL
LIN {X 0,Y 551.645,Z 406.184,A -85,B 0,C 180,E1 -3331.46,E2 -3331.46} C_VEL
LIN {X 0,Y 551.723,Z 403.81,A -85,B 0,C 180,E1 -3332.921,E2 -3332.921} C_VEL
LIN {X 0,Y 551.764,Z 400.895,A -85,B 0,C 180,E1 -3334.017,E2 -3334.017} C_VEL
LIN {X 0,Y 551.723,Z 396.948,A -85,B 0,C 180,E1 -3335.116,E2 -3335.116} C_VEL
LIN {X 0,Y 551.815,Z 391.122,A -85,B 0,C 180,E1 -3336.353,E2 -3336.353} C_VEL
LIN {X 0,Y 551.926,Z 384.235,A -85,B 0,C 180,E1 -3337.5,E2 -3337.5} C_VEL
LIN {X 0,Y 552.082,Z 375.99,A -85,B 0,C 180,E1 -3338.603,E2 -3338.603} C_VEL
LIN {X 0,Y 552.201,Z 367.538,A -85,B 0,C 180,E1 -3339.524,E2 -3339.524} C_VEL
LIN {X 0,Y 552.423,Z 357.09,A -85,B 0,C 180,E1 -3340.445,E2 -3340.445} C_VEL
LIN {X 0,Y 552.579,Z 345.343,A -85,B 0,C 180,E1 -3341.275,E2 -3341.275} C_VEL
LIN {X 0,Y 552.741,Z 333.483,A -85,B 0,C 180,E1 -3341.924,E2 -3341.924} C_VEL
LIN {X 0,Y 552.942,Z 321.159,A -85,B 0,C 180,E1 -3342.432,E2 -3342.432} C_VEL
LIN {X 0,Y 553.079,Z 308.507,A -85,B 0,C 180,E1 -3342.802,E2 -3342.802} C_VEL
LIN {X 0,Y 552.354,Z 302.494,A -85,B 0,C 180,E1 -3342.944,E2 -3342.944} C_VEL
LIN {X 0,Y 551.887,Z 299.529,A -85,B 0,C 180,E1 -3343.017,E2 -3343.017} C_VEL
LIN {X 0,Y 551.973,Z 289.414,A -85,B 0,C 180,E1 -3345.888,E2 -3345.888} C_VEL
LIN {X 0,Y 552.044,Z 279.69,A -85,B 0,C 180,E1 -3348.559,E2 -3348.559} C_VEL
LIN {X 0,Y 552.107,Z 269.977,A -85,B 0,C 180,E1 -3351.272,E2 -3351.272} C_VEL
LIN {X 0,Y 552.19,Z 260.375,A -85,B 0,C 180,E1 -3354.034,E2 -3354.034} C_VEL
LIN {X 0,Y 552.231,Z 252.197,A -85,B 0,C 180,E1 -3356.451,E2 -3356.451} C_VEL
LIN {X 0,Y 552.38,Z 242.953,A -85,B 0,C 180,E1 -3359.33,E2 -3359.33} C_VEL
LIN {X 0,Y 552.66,Z 234.201,A -85,B 0,C 180,E1 -3362.283,E2 -3362.283} C_VEL
LIN {X 0,Y 552.948,Z 227.355,A -85,B 0,C 180,E1 -3364.887,E2 -3364.887} C_VEL
LIN {X 0,Y 552.719,Z 223.123,A -85,B 0,C 180,E1 -3366.768,E2 -3366.768} C_VEL
LIN {X 0,Y 552.127,Z 219.713,A -85,B 0,C 180,E1 -3368.706,E2 -3368.706} C_VEL
LIN {X 0,Y 552.124,Z 219.714,A -85,B 0,C 180,E1 -3371.446,E2 -3371.446} C_VEL
LIN {X 0,Y 552.097,Z 219.716,A -85,B 0,C 180,E1 -3374.532,E2 -3374.532} C_VEL
LIN {X 0,Y 552.134,Z 219.711,A -85,B 0,C 180,E1 -3377.585,E2 -3377.585} C_VEL
LIN {X 0,Y 552.134,Z 219.713,A -85,B 0,C 180,E1 -3380.473,E2 -3380.473} C_VEL
LIN {X 0,Y 552.111,Z 219.715,A -85,B 0,C 180,E1 -3383.317,E2 -3383.317} C_VEL
LIN {X 0,Y 552.07,Z 219.72,A -85,B 0,C 180,E1 -3385.05,E2 -3385.05} C_VEL
LIN {X 0,Y 552.093,Z 220.236,A -85,B 0,C 180,E1 -3385.937,E2 -3385.937} C_VEL
LIN {X 0,Y 552.01,Z 222.804,A -85,B 0,C 180,E1 -3388.543,E2 -3388.543} C_VEL
LIN {X 0,Y 551.971,Z 225.765,A -85,B 0,C 180,E1 -3391.468,E2 -3391.468} C_VEL
LIN {X 0,Y 551.909,Z 228.728,A -85,B 0,C 180,E1 -3394.345,E2 -3394.345} C_VEL
LIN {X 0,Y 551.843,Z 231.239,A -85,B 0,C 180,E1 -3396.746,E2 -3396.746} C_VEL
LIN {X 0,Y 551.766,Z 233.708,A -85,B 0,C 180,E1 -3399.106,E2 -3399.106} C_VEL
LIN {X 0,Y 551.723,Z 236.156,A -85,B 0,C 180,E1 -3401.43,E2 -3401.43} C_VEL
LIN {X 0,Y 551.701,Z 238.655,A -85,B 0,C 180,E1 -3403.725,E2 -3403.725} C_VEL
LIN {X 0,Y 551.701,Z 241.203,A -85,B 0,C 180,E1 -3405.993,E2 -3405.993} C_VEL
LIN {X 0,Y 551.699,Z 243.678,A -85,B 0,C 180,E1 -3408.1,E2 -3408.1} C_VEL
LIN {X 0,Y 553.045,Z 252.56,A -85,B 0,C 180,E1 -3408.346,E2 -3408.346} C_VEL
LIN {X 0,Y 552.943,Z 264.593,A -85,B 0,C 180,E1 -3408.738,E2 -3408.738} C_VEL
LIN {X 0,Y 552.743,Z 276.72,A -85,B 0,C 180,E1 -3409.283,E2 -3409.283} C_VEL
LIN {X 0,Y 552.519,Z 287.782,A -85,B 0,C 180,E1 -3409.927,E2 -3409.927} C_VEL
LIN {X 0,Y 552.326,Z 299.069,A -85,B 0,C 180,E1 -3410.756,E2 -3410.756} C_VEL
LIN {X 0,Y 552.203,Z 308.154,A -85,B 0,C 180,E1 -3411.584,E2 -3411.584} C_VEL
LIN {X 0,Y 552.031,Z 316.476,A -85,B 0,C 180,E1 -3412.502,E2 -3412.502} C_VEL
LIN {X 0,Y 551.933,Z 324.337,A -85,B 0,C 180,E1 -3413.561,E2 -3413.561} C_VEL
LIN {X 0,Y 551.822,Z 330.174,A -85,B 0,C 180,E1 -3414.519,E2 -3414.519} C_VEL
LIN {X 0,Y 551.817,Z 335.601,A -85,B 0,C 180,E1 -3415.617,E2 -3415.617} C_VEL
LIN {X 0,Y 551.781,Z 339.854,A -85,B 0,C 180,E1 -3416.714,E2 -3416.714} C_VEL
LIN {X 0,Y 551.677,Z 343.051,A -85,B 0,C 180,E1 -3417.81,E2 -3417.81} C_VEL
LIN {X 0,Y 551.65,Z 344.643,A -85,B 0,C 180,E1 -3418.54,E2 -3418.54} C_VEL
LIN {X 0,Y 551.642,Z 345.829,A -85,B 0,C 180,E1 -3419.27,E2 -3419.27} C_VEL
LIN {X 0,Y 551.643,Z 346.58,A -85,B 0,C 180,E1 -3420,E2 -3420} C_VEL
LIN {X 0,Y 551.645,Z 346.916,A -85,B 0,C 180,E1 -3421.46,E2 -3421.46} C_VEL
LIN {X 0,Y 551.656,Z 346.511,A -85,B 0,C 180,E1 -3422.19,E2 -3422.19} C_VEL
LIN {X 0,Y 551.72,Z 345.677,A -85,B 0,C 180,E1 -3422.921,E2 -3422.921} C_VEL
LIN {X 0,Y 551.738,Z 344.437,A -85,B 0,C 180,E1 -3423.652,E2 -3423.652} C_VEL
LIN {X 0,Y 551.693,Z 341.804,A -85,B 0,C 180,E1 -3424.75,E2 -3424.75} C_VEL
LIN {X 0,Y 551.797,Z 338.161,A -85,B 0,C 180,E1 -3425.848,E2 -3425.848} C_VEL
LIN {X 0,Y 551.82,Z 333.4,A -85,B 0,C 180,E1 -3426.949,E2 -3426.949} C_VEL
LIN {X 0,Y 551.906,Z 326.259,A -85,B 0,C 180,E1 -3428.237,E2 -3428.237} C_VEL
LIN {X 0,Y 552.03,Z 318.46,A -85,B 0,C 180,E1 -3429.342,E2 -3429.342} C_VEL
LIN {X 0,Y 552.216,Z 308.702,A -85,B 0,C 180,E1 -3430.449,E2 -3430.449} C_VEL
LIN {X 0,Y 552.329,Z 298.337,A -85,B 0,C 180,E1 -3431.393,E2 -3431.393} C_VEL
LIN {X 0,Y 552.527,Z 287.076,A -85,B 0,C 180,E1 -3432.208,E2 -3432.208} C_VEL
LIN {X 0,Y 552.76,Z 275.776,A -85,B 0,C 180,E1 -3432.856,E2 -3432.856} C_VEL
LIN {X 0,Y 552.898,Z 264.254,A -85,B 0,C 180,E1 -3433.367,E2 -3433.367} C_VEL
LIN {X 0,Y 552.927,Z 250.978,A -85,B 0,C 180,E1 -3433.788,E2 -3433.788} C_VEL
LIN {X 0,Y 551.712,Z 243.687,A -85,B 0,C 180,E1 -3433.983,E2 -3433.983} C_VEL
LIN {X 0,Y 551.688,Z 239.818,A -85,B 0,C 180,E1 -3437.169,E2 -3437.169} C_VEL
LIN {X 0,Y 551.71,Z 236.365,A -85,B 0,C 180,E1 -3440.117,E2 -3440.117} C_VEL
LIN {X 0,Y 551.725,Z 233.688,A -85,B 0,C 180,E1 -3442.467,E2 -3442.467} C_VEL
LIN {X 0,Y 551.777,Z 230.362,A -85,B 0,C 180,E1 -3445.278,E2 -3445.278} C_VEL
LIN {X 0,Y 551.817,Z 227.063,A -85,B 0,C 180,E1 -3448.115,E2 -3448.115} C_VEL
LIN {X 0,Y 551.791,Z 226.702,A -85,B 0,C 180,E1 -3448.435,E2 -3448.435} C_VEL
LIN {X 0,Y 551.113,Z 226.082,A -85,B 0,C 180,E1 -3449.04,E2 -3449.04} C_VEL
LIN {X 0,Y 548.273,Z 225.218,A -85,B 0,C 180,E1 -3450.025,E2 -3450.025} C_VEL
LIN {X 0,Y 545.876,Z 224.487,A -85,B 0,C 180,E1 -3450.817,E2 -3450.817} C_VEL
LIN {X 0,Y 544.841,Z 223.85,A -85,B 0,C 180,E1 -3451.428,E2 -3451.428} C_VEL
LIN {X 0,Y 544.753,Z 223.617,A -85,B 0,C 180,E1 -3451.634,E2 -3451.634} C_VEL
LIN {X 0,Y 544.81,Z 220.626,A -85,B 0,C 180,E1 -3454.351,E2 -3454.351} C_VEL
LIN {X 0,Y 545.022,Z 220.593,A -85,B 0,C 180,E1 -3456.919,E2 -3456.919} C_VEL
LIN {X 0,Y 545.107,Z 220.582,A -85,B 0,C 180,E1 -3459.324,E2 -3459.324} C_VEL
LIN {X 0,Y 545.069,Z 220.59,A -85,B 0,C 180,E1 -3462.104,E2 -3462.104} C_VEL
LIN {X 0,Y 545.029,Z 220.594,A -85,B 0,C 180,E1 -3465.171,E2 -3465.171} C_VEL
LIN {X 0,Y 545.055,Z 220.588,A -85,B 0,C 180,E1 -3467.894,E2 -3467.894} C_VEL
LIN {X 0,Y 545.05,Z 220.591,A -85,B 0,C 180,E1 -3470.684,E2 -3470.684} C_VEL
LIN {X 0,Y 545.005,Z 220.593,A -85,B 0,C 180,E1 -3473.616,E2 -3473.616} C_VEL
LIN {X 0,Y 545.049,Z 220.592,A -85,B 0,C 180,E1 -3476.327,E2 -3476.327} C_VEL
LIN {X 0,Y 545.066,Z 220.587,A -85,B 0,C 180,E1 -3478.952,E2 -3478.952} C_VEL
LIN {X 0,Y 545.085,Z 220.585,A -85,B 0,C 180,E1 -3481.506,E2 -3481.506} C_VEL
LIN {X 0,Y 545.087,Z 220.585,A -85,B 0,C 180,E1 -3484.494,E2 -3484.494} C_VEL
LIN {X 0,Y 545.042,Z 220.592,A -85,B 0,C 180,E1 -3487.242,E2 -3487.242} C_VEL
LIN {X 0,Y 545.121,Z 220.579,A -85,B 0,C 180,E1 -3490.415,E2 -3490.415} C_VEL
LIN {X 0,Y 545.06,Z 220.59,A -85,B 0,C 180,E1 -3493.521,E2 -3493.521} C_VEL
LIN {X 0,Y 545.087,Z 220.584,A -85,B 0,C 180,E1 -3495.819,E2 -3495.819} C_VEL
LIN {X 0,Y 545.12,Z 220.585,A -85,B 0,C 180,E1 -3498.849,E2 -3498.849} C_VEL
LIN {X 0,Y 545.072,Z 220.587,A -85,B 0,C 180,E1 -3501.846,E2 -3501.846} C_VEL
LIN {X 0,Y 545.161,Z 220.574,A -85,B 0,C 180,E1 -3504.822,E2 -3504.822} C_VEL
LIN {X 0,Y 545.193,Z 220.577,A -85,B 0,C 180,E1 -3507.784,E2 -3507.784} C_VEL
LIN {X 0,Y 545.198,Z 220.573,A -85,B 0,C 180,E1 -3510,E2 -3510} C_VEL
LIN {X 0,Y 545.166,Z 220.575,A -85,B 0,C 180,E1 -3512.956,E2 -3512.956} C_VEL
LIN {X 0,Y 544.917,Z 220.613,A -85,B 0,C 180,E1 -3515.574,E2 -3515.574} C_VEL
LIN {X 0,Y 544.893,Z 226.532,A -85,B 0,C 180,E1 -3518.156,E2 -3518.156} C_VEL
LIN {X 0,Y 544.89,Z 233.903,A -85,B 0,C 180,E1 -3521.405,E2 -3521.405} C_VEL
LIN {X 0,Y 544.844,Z 241.253,A -85,B 0,C 180,E1 -3524.661,E2 -3524.661} C_VEL
LIN {X 0,Y 544.828,Z 247.178,A -85,B 0,C 180,E1 -3527.337,E2 -3527.337} C_VEL
LIN {X 0,Y 544.714,Z 253.816,A -85,B 0,C 180,E1 -3530.387,E2 -3530.387} C_VEL
LIN {X 0,Y 544.668,Z 259.185,A -85,B 0,C 180,E1 -3532.774,E2 -3532.774} C_VEL
LIN {X 0,Y 544.651,Z 264.805,A -85,B 0,C 180,E1 -3535.41,E2 -3535.41} C_VEL
LIN {X 0,Y 544.648,Z 267.617,A -85,B 0,C 180,E1 -3536.693,E2 -3536.693} C_VEL
LIN {X 0,Y 545.549,Z 275.771,A -85,B 0,C 180,E1 -3536.936,E2 -3536.936} C_VEL
LIN {X 0,Y 545.416,Z 287.367,A -85,B 0,C 180,E1 -3537.382,E2 -3537.382} C_VEL
LIN {X 0,Y 545.244,Z 297.885,A -85,B 0,C 180,E1 -3537.96,E2 -3537.96} C_VEL
LIN {X 0,Y 545.109,Z 306.681,A -85,B 0,C 180,E1 -3538.583,E2 -3538.583} C_VEL
LIN {X 0,Y 545.05,Z 313.511,A -85,B 0,C 180,E1 -3539.174,E2 -3539.174} C_VEL
LIN {X 0,Y 544.945,Z 319.381,A -85,B 0,C 180,E1 -3539.77,E2 -3539.77} C_VEL
LIN {X 0,Y 544.8,Z 326.304,A -85,B 0,C 180,E1 -3540.634,E2 -3540.634} C_VEL
LIN {X 0,Y 544.752,Z 332.657,A -85,B 0,C 180,E1 -3541.626,E2 -3541.626} C_VEL
LIN {X 0,Y 544.663,Z 336.58,A -85,B 0,C 180,E1 -3542.377,E2 -3542.377} C_VEL
LIN {X 0,Y 544.648,Z 340.456,A -85,B 0,C 180,E1 -3543.316,E2 -3543.316} C_VEL
LIN {X 0,Y 544.605,Z 344.174,A -85,B 0,C 180,E1 -3544.598,E2 -3544.598} C_VEL
LIN {X 0,Y 544.554,Z 345.972,A -85,B 0,C 180,E1 -3545.602,E2 -3545.602} C_VEL
LIN {X 0,Y 544.558,Z 346.943,A -85,B 0,C 180,E1 -3546.854,E2 -3546.854} C_VEL
LIN {X 0,Y 544.528,Z 346.259,A -85,B 0,C 180,E1 -3548.281,E2 -3548.281} C_VEL
LIN {X 0,Y 544.561,Z 344.732,A -85,B 0,C 180,E1 -3549.254,E2 -3549.254} C_VEL
LIN {X 0,Y 544.625,Z 341.652,A -85,B 0,C 180,E1 -3550.416,E2 -3550.416} C_VEL
LIN {X 0,Y 544.649,Z 339.037,A -85,B 0,C 180,E1 -3551.155,E2 -3551.155} C_VEL
LIN {X 0,Y 544.697,Z 334.466,A -85,B 0,C 180,E1 -3552.139,E2 -3552.139} C_VEL
LIN {X 0,Y 544.773,Z 328.496,A -85,B 0,C 180,E1 -3553.137,E2 -3553.137} C_VEL
LIN {X 0,Y 544.861,Z 322.701,A -85,B 0,C 180,E1 -3553.921,E2 -3553.921} C_VEL
LIN {X 0,Y 544.952,Z 316.139,A -85,B 0,C 180,E1 -3554.657,E2 -3554.657} C_VEL
LIN {X 0,Y 545.07,Z 309.251,A -85,B 0,C 180,E1 -3555.298,E2 -3555.298} C_VEL
LIN {X 0,Y 545.218,Z 301.551,A -85,B 0,C 180,E1 -3555.887,E2 -3555.887} C_VEL
LIN {X 0,Y 545.323,Z 293.341,A -85,B 0,C 180,E1 -3556.397,E2 -3556.397} C_VEL
LIN {X 0,Y 545.458,Z 285.127,A -85,B 0,C 180,E1 -3556.804,E2 -3556.804} C_VEL
LIN {X 0,Y 545.532,Z 274.941,A -85,B 0,C 180,E1 -3557.179,E2 -3557.179} C_VEL
LIN {X 0,Y 544.649,Z 267.591,A -85,B 0,C 180,E1 -3557.403,E2 -3557.403} C_VEL
LIN {X 0,Y 544.667,Z 262.408,A -85,B 0,C 180,E1 -3559.822,E2 -3559.822} C_VEL
LIN {X 0,Y 544.701,Z 257.867,A -85,B 0,C 180,E1 -3561.911,E2 -3561.911} C_VEL
LIN {X 0,Y 544.727,Z 251.304,A -85,B 0,C 180,E1 -3564.961,E2 -3564.961} C_VEL
LIN {X 0,Y 544.772,Z 246.213,A -85,B 0,C 180,E1 -3567.191,E2 -3567.191} C_VEL
LIN {X 0,Y 544.799,Z 240.311,A -85,B 0,C 180,E1 -3569.805,E2 -3569.805} C_VEL
LIN {X 0,Y 544.792,Z 234.512,A -85,B 0,C 180,E1 -3572.328,E2 -3572.328} C_VEL
LIN {X 0,Y 544.857,Z 228.632,A -85,B 0,C 180,E1 -3574.807,E2 -3574.807} C_VEL
LIN {X 0,Y 544.855,Z 220.621,A -85,B 0,C 180,E1 -3578.1,E2 -3578.1} C_VEL
LIN {X 0,Y 545.12,Z 220.584,A -85,B 0,C 180,E1 -3580.415,E2 -3580.415} C_VEL
LIN {X 0,Y 545.067,Z 220.593,A -85,B 0,C 180,E1 -3583.521,E2 -3583.521} C_VEL
LIN {X 0,Y 545.094,Z 220.59,A -85,B 0,C 180,E1 -3585.82,E2 -3585.82} C_VEL
LIN {X 0,Y 545.122,Z 220.584,A -85,B 0,C 180,E1 -3588.849,E2 -3588.849} C_VEL
LIN {X 0,Y 545.132,Z 220.585,A -85,B 0,C 180,E1 -3591.847,E2 -3591.847} C_VEL
LIN {X 0,Y 545.203,Z 220.573,A -85,B 0,C 180,E1 -3594.823,E2 -3594.823} C_VEL
LIN {X 0,Y 545.199,Z 220.577,A -85,B 0,C 180,E1 -3597.784,E2 -3597.784} C_VEL
LIN {X 0,Y 545.212,Z 220.572,A -85,B 0,C 180,E1 -3600.739,E2 -3600.739} C_VEL
LIN {X 0,Y 545.173,Z 220.577,A -85,B 0,C 180,E1 -3602.956,E2 -3602.956} C_VEL
LIN {X 0,Y 545.164,Z 220.58,A -85,B 0,C 180,E1 -3605.92,E2 -3605.92} C_VEL
LIN {X 0,Y 545.113,Z 220.584,A -85,B 0,C 180,E1 -3608.9,E2 -3608.9} C_VEL
LIN {X 0,Y 545.138,Z 220.583,A -85,B 0,C 180,E1 -3611.904,E2 -3611.904} C_VEL
LIN {X 0,Y 545.089,Z 220.587,A -85,B 0,C 180,E1 -3614.943,E2 -3614.943} C_VEL
LIN {X 0,Y 545.074,Z 220.591,A -85,B 0,C 180,E1 -3618.026,E2 -3618.026} C_VEL
LIN {X 0,Y 545.096,Z 220.589,A -85,B 0,C 180,E1 -3620.372,E2 -3620.372} C_VEL
LIN {X 0,Y 545.082,Z 220.589,A -85,B 0,C 180,E1 -3623.559,E2 -3623.559} C_VEL
LIN {X 0,Y 545.072,Z 220.591,A -85,B 0,C 180,E1 -3626.001,E2 -3626.001} C_VEL
LIN {X 0,Y 545.092,Z 220.589,A -85,B 0,C 180,E1 -3628.748,E2 -3628.748} C_VEL
LIN {X 0,Y 545.057,Z 220.592,A -85,B 0,C 180,E1 -3631.915,E2 -3631.915} C_VEL
LIN {X 0,Y 545.062,Z 220.593,A -85,B 0,C 180,E1 -3634.565,E2 -3634.565} C_VEL
LIN {X 0,Y 545.039,Z 220.594,A -85,B 0,C 180,E1 -3637.304,E2 -3637.304} C_VEL
LIN {X 0,Y 545.068,Z 220.59,A -85,B 0,C 180,E1 -3640.143,E2 -3640.143} C_VEL
LIN {X 0,Y 545.081,Z 220.59,A -85,B 0,C 180,E1 -3643.107,E2 -3643.107} C_VEL
LIN {X 0,Y 545.051,Z 220.594,A -85,B 0,C 180,E1 -3646.226,E2 -3646.226} C_VEL
LIN {X 0,Y 545.084,Z 220.59,A -85,B 0,C 180,E1 -3648.885,E2 -3648.885} C_VEL
LIN {X 0,Y 545.085,Z 220.589,A -85,B 0,C 180,E1 -3650.819,E2 -3650.819} C_VEL
LIN {X 0,Y 545.066,Z 220.669,A -85,B 0,C 180,E1 -3652.291,E2 -3652.291} C_VEL
LIN {X 0,Y 545.903,Z 225.791,A -85,B 0,C 180,E1 -3654.201,E2 -3654.201} C_VEL
LIN {X 0,Y 545.884,Z 232.091,A -85,B 0,C 180,E1 -3656.385,E2 -3656.385} C_VEL
LIN {X 0,Y 545.629,Z 241.017,A -85,B 0,C 180,E1 -3659.368,E2 -3659.368} C_VEL
LIN {X 0,Y 545.385,Z 250.349,A -85,B 0,C 180,E1 -3662.36,E2 -3662.36} C_VEL
LIN {X 0,Y 545.236,Z 259.616,A -85,B 0,C 180,E1 -3665.234,E2 -3665.234} C_VEL
LIN {X 0,Y 545.144,Z 269.323,A -85,B 0,C 180,E1 -3668.16,E2 -3668.16} C_VEL
LIN {X 0,Y 544.996,Z 279.624,A -85,B 0,C 180,E1 -3671.193,E2 -3671.193} C_VEL
LIN {X 0,Y 544.899,Z 289.158,A -85,B 0,C 180,E1 -3673.901,E2 -3673.901} C_VEL
LIN {X 0,Y 544.803,Z 298.648,A -85,B 0,C 180,E1 -3676.573,E2 -3676.573} C_VEL
LIN {X 0,Y 544.802,Z 299.494,A -85,B 0,C 180,E1 -3676.811,E2 -3676.811} C_VEL
LIN {X 0,Y 546.178,Z 309.436,A -85,B 0,C 180,E1 -3677.057,E2 -3677.057} C_VEL
LIN {X 0,Y 545.976,Z 322.475,A -85,B 0,C 180,E1 -3677.454,E2 -3677.454} C_VEL
LIN {X 0,Y 545.784,Z 333.49,A -85,B 0,C 180,E1 -3677.922,E2 -3677.922} C_VEL
LIN {X 0,Y 545.583,Z 345.608,A -85,B 0,C 180,E1 -3678.596,E2 -3678.596} C_VEL
LIN {X 0,Y 545.419,Z 357.092,A -85,B 0,C 180,E1 -3679.419,E2 -3679.419} C_VEL
LIN {X 0,Y 545.165,Z 367.54,A -85,B 0,C 180,E1 -3680.352,E2 -3680.352} C_VEL
LIN {X 0,Y 545.029,Z 375.992,A -85,B 0,C 180,E1 -3681.285,E2 -3681.285} C_VEL
LIN {X 0,Y 544.859,Z 384.236,A -85,B 0,C 180,E1 -3682.403,E2 -3682.403} C_VEL
LIN {X 0,Y 544.734,Z 391.616,A -85,B 0,C 180,E1 -3683.655,E2 -3683.655} C_VEL
LIN {X 0,Y 544.653,Z 396.95,A -85,B 0,C 180,E1 -3684.818,E2 -3684.818} C_VEL
LIN {X 0,Y 544.684,Z 400.895,A -85,B 0,C 180,E1 -3685.931,E2 -3685.931} C_VEL
LIN {X 0,Y 544.65,Z 403.807,A -85,B 0,C 180,E1 -3687.041,E2 -3687.041} C_VEL
LIN {X 0,Y 544.546,Z 406.183,A -85,B 0,C 180,E1 -3688.521,E2 -3688.521} C_VEL
LIN {X 0,Y 544.541,Z 407,A -85,B 0,C 180,E1 -3690,E2 -3690} C_VEL
LIN {X 0,Y 544.546,Z 406.184,A -85,B 0,C 180,E1 -3691.479,E2 -3691.479} C_VEL
LIN {X 0,Y 544.65,Z 403.81,A -85,B 0,C 180,E1 -3692.959,E2 -3692.959} C_VEL
LIN {X 0,Y 544.684,Z 400.895,A -85,B 0,C 180,E1 -3694.07,E2 -3694.07} C_VEL
LIN {X 0,Y 544.653,Z 396.948,A -85,B 0,C 180,E1 -3695.182,E2 -3695.182} C_VEL
LIN {X 0,Y 544.73,Z 391.641,A -85,B 0,C 180,E1 -3696.34,E2 -3696.34} C_VEL
LIN {X 0,Y 544.836,Z 385.465,A -85,B 0,C 180,E1 -3697.412,E2 -3697.412} C_VEL
LIN {X 0,Y 545.007,Z 377.476,A -85,B 0,C 180,E1 -3698.528,E2 -3698.528} C_VEL
LIN {X 0,Y 545.142,Z 369.331,A -85,B 0,C 180,E1 -3699.461,E2 -3699.461} C_VEL
LIN {X 0,Y 545.37,Z 359.395,A -85,B 0,C 180,E1 -3700.394,E2 -3700.394} C_VEL
LIN {X 0,Y 545.525,Z 349.589,A -85,B 0,C 180,E1 -3701.142,E2 -3701.142} C_VEL
LIN {X 0,Y 545.69,Z 338.619,A -85,B 0,C 180,E1 -3701.815,E2 -3701.815} C_VEL
LIN {X 0,Y 545.894,Z 326.096,A -85,B 0,C 180,E1 -3702.406,E2 -3702.406} C_VEL
LIN {X 0,Y 546.131,Z 313.078,A -85,B 0,C 180,E1 -3702.849,E2 -3702.849} C_VEL
LIN {X 0,Y 545.898,Z 306.351,A -85,B 0,C 180,E1 -3703.021,E2 -3703.021} C_VEL
LIN {X 0,Y 544.802,Z 299.485,A -85,B 0,C 180,E1 -3703.19,E2 -3703.19} C_VEL
LIN {X 0,Y 544.898,Z 288.969,A -85,B 0,C 180,E1 -3706.1,E2 -3706.1} C_VEL
LIN {X 0,Y 544.972,Z 279.235,A -85,B 0,C 180,E1 -3708.808,E2 -3708.808} C_VEL
LIN {X 0,Y 545.091,Z 268.222,A -85,B 0,C 180,E1 -3711.957,E2 -3711.957} C_VEL
LIN {X 0,Y 545.132,Z 258.624,A -85,B 0,C 180,E1 -3714.772,E2 -3714.772} C_VEL
LIN {X 0,Y 545.272,Z 249.274,A -85,B 0,C 180,E1 -3717.646,E2 -3717.646} C_VEL
LIN {X 0,Y 545.465,Z 240.222,A -85,B 0,C 180,E1 -3720.623,E2 -3720.623} C_VEL
LIN {X 0,Y 545.8,Z 233.099,A -85,B 0,C 180,E1 -3723.178,E2 -3723.178} C_VEL
LIN {X 0,Y 545.991,Z 227.611,A -85,B 0,C 180,E1 -3725.397,E2 -3725.397} C_VEL
LIN {X 0,Y 545.646,Z 223.717,A -85,B 0,C 180,E1 -3727.256,E2 -3727.256} C_VEL
LIN {X 0,Y 545.096,Z 220.59,A -85,B 0,C 180,E1 -3729.121,E2 -3729.121} C_VEL
LIN {X 0,Y 545.081,Z 220.59,A -85,B 0,C 180,E1 -3732.103,E2 -3732.103} C_VEL
LIN {X 0,Y 545.039,Z 220.596,A -85,B 0,C 180,E1 -3735.17,E2 -3735.17} C_VEL
LIN {X 0,Y 545.081,Z 220.591,A -85,B 0,C 180,E1 -3737.897,E2 -3737.897} C_VEL
LIN {X 0,Y 545.084,Z 220.59,A -85,B 0,C 180,E1 -3740.819,E2 -3740.819} C_VEL
LIN {X 0,Y 545.046,Z 220.595,A -85,B 0,C 180,E1 -3743.62,E2 -3743.62} C_VEL
LIN {X 0,Y 545.046,Z 220.938,A -85,B 0,C 180,E1 -3745.613,E2 -3745.613} C_VEL
LIN {X 0,Y 544.981,Z 223.519,A -85,B 0,C 180,E1 -3748.335,E2 -3748.335} C_VEL
LIN {X 0,Y 544.922,Z 226.644,A -85,B 0,C 180,E1 -3751.497,E2 -3751.497} C_VEL
LIN {X 0,Y 544.861,Z 229.984,A -85,B 0,C 180,E1 -3754.808,E2 -3754.808} C_VEL
LIN {X 0,Y 544.768,Z 233.352,A -85,B 0,C 180,E1 -3758.03,E2 -3758.03} C_VEL
LIN {X 0,Y 544.664,Z 236.623,A -85,B 0,C 180,E1 -3761.181,E2 -3761.181} C_VEL
LIN {X 0,Y 544.66,Z 239.094,A -85,B 0,C 180,E1 -3763.508,E2 -3763.508} C_VEL
LIN {X 0,Y 544.636,Z 241.632,A -85,B 0,C 180,E1 -3765.808,E2 -3765.808} C_VEL
LIN {X 0,Y 544.645,Z 244.067,A -85,B 0,C 180,E1 -3767.943,E2 -3767.943} C_VEL
LIN {X 0,Y 546.13,Z 252.969,A -85,B 0,C 180,E1 -3768.19,E2 -3768.19} C_VEL
LIN {X 0,Y 546,Z 265.55,A -85,B 0,C 180,E1 -3768.615,E2 -3768.615} C_VEL
LIN {X 0,Y 545.791,Z 277.055,A -85,B 0,C 180,E1 -3769.145,E2 -3769.145} C_VEL
LIN {X 0,Y 545.538,Z 288.042,A -85,B 0,C 180,E1 -3769.797,E2 -3769.797} C_VEL
LIN {X 0,Y 545.318,Z 299.239,A -85,B 0,C 180,E1 -3770.636,E2 -3770.636} C_VEL
LIN {X 0,Y 545.19,Z 308.284,A -85,B 0,C 180,E1 -3771.475,E2 -3771.475} C_VEL
LIN {X 0,Y 544.981,Z 316.586,A -85,B 0,C 180,E1 -3772.404,E2 -3772.404} C_VEL
LIN {X 0,Y 544.869,Z 324.929,A -85,B 0,C 180,E1 -3773.553,E2 -3773.553} C_VEL
LIN {X 0,Y 544.765,Z 330.248,A -85,B 0,C 180,E1 -3774.448,E2 -3774.448} C_VEL
LIN {X 0,Y 544.736,Z 335.66,A -85,B 0,C 180,E1 -3775.56,E2 -3775.56} C_VEL
LIN {X 0,Y 544.708,Z 339.899,A -85,B 0,C 180,E1 -3776.672,E2 -3776.672} C_VEL
LIN {X 0,Y 544.592,Z 343.083,A -85,B 0,C 180,E1 -3777.781,E2 -3777.781} C_VEL
LIN {X 0,Y 544.551,Z 344.669,A -85,B 0,C 180,E1 -3778.521,E2 -3778.521} C_VEL
LIN {X 0,Y 544.542,Z 345.847,A -85,B 0,C 180,E1 -3779.261,E2 -3779.261} C_VEL
LIN {X 0,Y 544.541,Z 346.941,A -85,B 0,C 180,E1 -3780.74,E2 -3780.74} C_VEL
LIN {X 0,Y 544.571,Z 346.5,A -85,B 0,C 180,E1 -3782.219,E2 -3782.219} C_VEL
LIN {X 0,Y 544.647,Z 345.656,A -85,B 0,C 180,E1 -3782.959,E2 -3782.959} C_VEL
LIN {X 0,Y 544.653,Z 344.409,A -85,B 0,C 180,E1 -3783.699,E2 -3783.699} C_VEL
LIN {X 0,Y 544.602,Z 341.765,A -85,B 0,C 180,E1 -3784.812,E2 -3784.812} C_VEL
LIN {X 0,Y 544.705,Z 338.109,A -85,B 0,C 180,E1 -3785.925,E2 -3785.925} C_VEL
LIN {X 0,Y 544.735,Z 333.333,A -85,B 0,C 180,E1 -3787.04,E2 -3787.04} C_VEL
LIN {X 0,Y 544.853,Z 326.177,A -85,B 0,C 180,E1 -3788.344,E2 -3788.344} C_VEL
LIN {X 0,Y 544.961,Z 318.35,A -85,B 0,C 180,E1 -3789.464,E2 -3789.464} C_VEL
LIN {X 0,Y 545.198,Z 308.569,A -85,B 0,C 180,E1 -3790.585,E2 -3790.585} C_VEL
LIN {X 0,Y 545.316,Z 298.998,A -85,B 0,C 180,E1 -3791.474,E2 -3791.474} C_VEL
LIN {X 0,Y 545.523,Z 288.33,A -85,B 0,C 180,E1 -3792.273,E2 -3792.273} C_VEL
LIN {X 0,Y 545.782,Z 277.337,A -85,B 0,C 180,E1 -3792.929,E2 -3792.929} C_VEL
LIN {X 0,Y 545.942,Z 265.145,A -85,B 0,C 180,E1 -3793.493,E2 -3793.493} C_VEL
LIN {X 0,Y 546.075,Z 252.325,A -85,B 0,C 180,E1 -3793.917,E2 -3793.917} C_VEL
LIN {X 0,Y 544.609,Z 243.848,A -85,B 0,C 180,E1 -3794.169,E2 -3794.169} C_VEL
LIN {X 0,Y 544.618,Z 240.17,A -85,B 0,C 180,E1 -3797.266,E2 -3797.266} C_VEL
LIN {X 0,Y 544.625,Z 236.565,A -85,B 0,C 180,E1 -3800.391,E2 -3800.391} C_VEL
LIN {X 0,Y 544.64,Z 233.867,A -85,B 0,C 180,E1 -3802.776,E2 -3802.776} C_VEL
LIN {X 0,Y 544.729,Z 230.08,A -85,B 0,C 180,E1 -3806.019,E2 -3806.019} C_VEL
LIN {X 0,Y 544.705,Z 227.025,A -85,B 0,C 180,E1 -3808.673,E2 -3808.673} C_VEL
LIN {X 0,Y 544.753,Z 223.617,A -85,B 0,C 180,E1 -3811.634,E2 -3811.634} C_VEL
LIN {X 0,Y 544.074,Z 222.97,A -85,B 0,C 180,E1 -3812.247,E2 -3812.247} C_VEL
LIN {X 0,Y 541.23,Z 222.085,A -85,B 0,C 180,E1 -3813.245,E2 -3813.245} C_VEL
LIN {X 0,Y 538.858,Z 221.657,A -85,B 0,C 180,E1 -3814.05,E2 -3814.05} C_VEL
LIN {X 0,Y 537.875,Z 221.509,A -85,B 0,C 180,E1 -3814.671,E2 -3814.671} C_VEL
LIN {X 0,Y 537.813,Z 221.497,A -85,B 0,C 180,E1 -3814.882,E2 -3814.882} C_VEL
LIN {X 0,Y 537.979,Z 221.469,A -85,B 0,C 180,E1 -3817.166,E2 -3817.166} C_VEL
LIN {X 0,Y 538.029,Z 221.469,A -85,B 0,C 180,E1 -3819.797,E2 -3819.797} C_VEL
LIN {X 0,Y 538.005,Z 221.466,A -85,B 0,C 180,E1 -3822.788,E2 -3822.788} C_VEL
LIN {X 0,Y 538.002,Z 221.469,A -85,B 0,C 180,E1 -3825.137,E2 -3825.137} C_VEL
LIN {X 0,Y 538.003,Z 221.465,A -85,B 0,C 180,E1 -3828.224,E2 -3828.224} C_VEL
LIN {X 0,Y 537.992,Z 221.472,A -85,B 0,C 180,E1 -3831.167,E2 -3831.167} C_VEL
LIN {X 0,Y 537.959,Z 221.471,A -85,B 0,C 180,E1 -3834.094,E2 -3834.094} C_VEL
LIN {X 0,Y 538.035,Z 221.467,A -85,B 0,C 180,E1 -3836.727,E2 -3836.727} C_VEL
LIN {X 0,Y 538.01,Z 221.465,A -85,B 0,C 180,E1 -3839.56,E2 -3839.56} C_VEL
LIN {X 0,Y 538.024,Z 221.468,A -85,B 0,C 180,E1 -3841.949,E2 -3841.949} C_VEL
LIN {X 0,Y 538.064,Z 221.46,A -85,B 0,C 180,E1 -3844.466,E2 -3844.466} C_VEL
LIN {X 0,Y 538.019,Z 221.465,A -85,B 0,C 180,E1 -3846.928,E2 -3846.928} C_VEL
LIN {X 0,Y 538.085,Z 221.456,A -85,B 0,C 180,E1 -3850.148,E2 -3850.148} C_VEL
LIN {X 0,Y 538.008,Z 221.471,A -85,B 0,C 180,E1 -3853.298,E2 -3853.298} C_VEL
LIN {X 0,Y 538.059,Z 221.46,A -85,B 0,C 180,E1 -3855.63,E2 -3855.63} C_VEL
LIN {X 0,Y 538.08,Z 221.462,A -85,B 0,C 180,E1 -3858.701,E2 -3858.701} C_VEL
LIN {X 0,Y 538.043,Z 221.462,A -85,B 0,C 180,E1 -3861.739,E2 -3861.739} C_VEL
LIN {X 0,Y 538.121,Z 221.452,A -85,B 0,C 180,E1 -3864.754,E2 -3864.754} C_VEL
LIN {X 0,Y 538.164,Z 221.452,A -85,B 0,C 180,E1 -3867.755,E2 -3867.755} C_VEL
LIN {X 0,Y 538.167,Z 221.448,A -85,B 0,C 180,E1 -3870,E2 -3870} C_VEL
LIN {X 0,Y 538.134,Z 221.452,A -85,B 0,C 180,E1 -3872.994,E2 -3872.994} C_VEL
LIN {X 0,Y 537.849,Z 221.561,A -85,B 0,C 180,E1 -3875.671,E2 -3875.671} C_VEL
LIN {X 0,Y 537.822,Z 227.527,A -85,B 0,C 180,E1 -3878.264,E2 -3878.264} C_VEL
LIN {X 0,Y 537.831,Z 234.789,A -85,B 0,C 180,E1 -3881.463,E2 -3881.463} C_VEL
LIN {X 0,Y 537.788,Z 242.114,A -85,B 0,C 180,E1 -3884.746,E2 -3884.746} C_VEL
LIN {X 0,Y 537.745,Z 248.164,A -85,B 0,C 180,E1 -3887.493,E2 -3887.493} C_VEL
LIN {X 0,Y 537.664,Z 253.349,A -85,B 0,C 180,E1 -3889.868,E2 -3889.868} C_VEL
LIN {X 0,Y 537.604,Z 258.701,A -85,B 0,C 180,E1 -3892.279,E2 -3892.279} C_VEL
LIN {X 0,Y 537.585,Z 263.966,A -85,B 0,C 180,E1 -3894.73,E2 -3894.73} C_VEL
LIN {X 0,Y 537.581,Z 267.831,A -85,B 0,C 180,E1 -3896.548,E2 -3896.548} C_VEL
LIN {X 0,Y 538.583,Z 276.257,A -85,B 0,C 180,E1 -3896.808,E2 -3896.808} C_VEL
LIN {X 0,Y 538.428,Z 287.828,A -85,B 0,C 180,E1 -3897.262,E2 -3897.262} C_VEL
LIN {X 0,Y 538.252,Z 298.326,A -85,B 0,C 180,E1 -3897.848,E2 -3897.848} C_VEL
LIN {X 0,Y 538.114,Z 307.005,A -85,B 0,C 180,E1 -3898.47,E2 -3898.47} C_VEL
LIN {X 0,Y 538.026,Z 314.113,A -85,B 0,C 180,E1 -3899.095,E2 -3899.095} C_VEL
LIN {X 0,Y 537.895,Z 320.523,A -85,B 0,C 180,E1 -3899.769,E2 -3899.769} C_VEL
LIN {X 0,Y 537.758,Z 327.297,A -85,B 0,C 180,E1 -3900.644,E2 -3900.644} C_VEL
LIN {X 0,Y 537.7,Z 332.796,A -85,B 0,C 180,E1 -3901.522,E2 -3901.522} C_VEL
LIN {X 0,Y 537.6,Z 337.284,A -85,B 0,C 180,E1 -3902.411,E2 -3902.411} C_VEL
LIN {X 0,Y 537.569,Z 340.844,A -85,B 0,C 180,E1 -3903.305,E2 -3903.305} C_VEL
LIN {X 0,Y 537.513,Z 344.347,A -85,B 0,C 180,E1 -3904.54,E2 -3904.54} C_VEL
LIN {X 0,Y 537.492,Z 345.564,A -85,B 0,C 180,E1 -3905.122,E2 -3905.122} C_VEL
LIN {X 0,Y 537.47,Z 346.77,A -85,B 0,C 180,E1 -3906.045,E2 -3906.045} C_VEL
LIN {X 0,Y 537.446,Z 347.206,A -85,B 0,C 180,E1 -3907.091,E2 -3907.091} C_VEL
LIN {X 0,Y 537.433,Z 346.457,A -85,B 0,C 180,E1 -3908.314,E2 -3908.314} C_VEL
LIN {X 0,Y 537.493,Z 344.435,A -85,B 0,C 180,E1 -3909.515,E2 -3909.515} C_VEL
LIN {X 0,Y 537.555,Z 342.565,A -85,B 0,C 180,E1 -3910.26,E2 -3910.26} C_VEL
LIN {X 0,Y 537.574,Z 338.857,A -85,B 0,C 180,E1 -3911.316,E2 -3911.316} C_VEL
LIN {X 0,Y 537.643,Z 334.199,A -85,B 0,C 180,E1 -3912.314,E2 -3912.314} C_VEL
LIN {X 0,Y 537.721,Z 329.466,A -85,B 0,C 180,E1 -3913.127,E2 -3913.127} C_VEL
LIN {X 0,Y 537.82,Z 322.769,A -85,B 0,C 180,E1 -3914.051,E2 -3914.051} C_VEL
LIN {X 0,Y 537.925,Z 316.507,A -85,B 0,C 180,E1 -3914.759,E2 -3914.759} C_VEL
LIN {X 0,Y 538.084,Z 308.561,A -85,B 0,C 180,E1 -3915.494,E2 -3915.494} C_VEL
LIN {X 0,Y 538.209,Z 301.121,A -85,B 0,C 180,E1 -3916.056,E2 -3916.056} C_VEL
LIN {X 0,Y 538.348,Z 293.108,A -85,B 0,C 180,E1 -3916.551,E2 -3916.551} C_VEL
LIN {X 0,Y 538.475,Z 284.754,A -85,B 0,C 180,E1 -3916.962,E2 -3916.962} C_VEL
LIN {X 0,Y 538.571,Z 275.162,A -85,B 0,C 180,E1 -3917.316,E2 -3917.316} C_VEL
LIN {X 0,Y 537.576,Z 267.872,A -85,B 0,C 180,E1 -3917.552,E2 -3917.552} C_VEL
LIN {X 0,Y 537.626,Z 261.718,A -85,B 0,C 180,E1 -3920.468,E2 -3920.468} C_VEL
LIN {X 0,Y 537.635,Z 256.061,A -85,B 0,C 180,E1 -3923.036,E2 -3923.036} C_VEL
LIN {X 0,Y 537.73,Z 248.907,A -85,B 0,C 180,E1 -3926.257,E2 -3926.257} C_VEL
LIN {X 0,Y 537.695,Z 241.997,A -85,B 0,C 180,E1 -3929.352,E2 -3929.352} C_VEL
LIN {X 0,Y 537.735,Z 236.086,A -85,B 0,C 180,E1 -3931.933,E2 -3931.933} C_VEL
LIN {X 0,Y 537.771,Z 228.231,A -85,B 0,C 180,E1 -3935.279,E2 -3935.279} C_VEL
LIN {X 0,Y 537.819,Z 221.498,A -85,B 0,C 180,E1 -3938.095,E2 -3938.095} C_VEL
LIN {X 0,Y 538.042,Z 221.467,A -85,B 0,C 180,E1 -3940.146,E2 -3940.146} C_VEL
LIN {X 0,Y 538.031,Z 221.468,A -85,B 0,C 180,E1 -3942.516,E2 -3942.516} C_VEL
LIN {X 0,Y 538.064,Z 221.464,A -85,B 0,C 180,E1 -3945.631,E2 -3945.631} C_VEL
LIN {X 0,Y 538.082,Z 221.461,A -85,B 0,C 180,E1 -3948.701,E2 -3948.701} C_VEL
LIN {X 0,Y 538.089,Z 221.462,A -85,B 0,C 180,E1 -3951.74,E2 -3951.74} C_VEL
LIN {X 0,Y 538.158,Z 221.451,A -85,B 0,C 180,E1 -3954.755,E2 -3954.755} C_VEL
LIN {X 0,Y 538.171,Z 221.452,A -85,B 0,C 180,E1 -3957.755,E2 -3957.755} C_VEL
LIN {X 0,Y 538.183,Z 221.448,A -85,B 0,C 180,E1 -3960.748,E2 -3960.748} C_VEL
LIN {X 0,Y 538.139,Z 221.453,A -85,B 0,C 180,E1 -3962.994,E2 -3962.994} C_VEL
LIN {X 0,Y 538.116,Z 221.459,A -85,B 0,C 180,E1 -3965.997,E2 -3965.997} C_VEL
LIN {X 0,Y 538.064,Z 221.462,A -85,B 0,C 180,E1 -3969.018,E2 -3969.018} C_VEL
LIN {X 0,Y 538.087,Z 221.462,A -85,B 0,C 180,E1 -3972.062,E2 -3972.062} C_VEL
LIN {X 0,Y 538.048,Z 221.465,A -85,B 0,C 180,E1 -3975.144,E2 -3975.144} C_VEL
LIN {X 0,Y 538.028,Z 221.467,A -85,B 0,C 180,E1 -3978.27,E2 -3978.27} C_VEL
LIN {X 0,Y 538.041,Z 221.466,A -85,B 0,C 180,E1 -3980.651,E2 -3980.651} C_VEL
LIN {X 0,Y 538.009,Z 221.472,A -85,B 0,C 180,E1 -3983.878,E2 -3983.878} C_VEL
LIN {X 0,Y 538.037,Z 221.467,A -85,B 0,C 180,E1 -3986.367,E2 -3986.367} C_VEL
LIN {X 0,Y 538.032,Z 221.467,A -85,B 0,C 180,E1 -3988.933,E2 -3988.933} C_VEL
LIN {X 0,Y 538.012,Z 221.469,A -85,B 0,C 180,E1 -3991.887,E2 -3991.887} C_VEL
LIN {X 0,Y 538.012,Z 221.471,A -85,B 0,C 180,E1 -3994.617,E2 -3994.617} C_VEL
LIN {X 0,Y 538.007,Z 221.47,A -85,B 0,C 180,E1 -3997.17,E2 -3997.17} C_VEL
LIN {X 0,Y 538.025,Z 221.467,A -85,B 0,C 180,E1 -3999.797,E2 -3999.797} C_VEL
LIN {X 0,Y 538.021,Z 221.469,A -85,B 0,C 180,E1 -4002.786,E2 -4002.786} C_VEL
LIN {X 0,Y 538.021,Z 221.468,A -85,B 0,C 180,E1 -4005.927,E2 -4005.927} C_VEL
LIN {X 0,Y 538.033,Z 221.466,A -85,B 0,C 180,E1 -4008.227,E2 -4008.227} C_VEL
LIN {X 0,Y 538.017,Z 221.47,A -85,B 0,C 180,E1 -4011.17,E2 -4011.17} C_VEL
LIN {X 0,Y 538.037,Z 221.578,A -85,B 0,C 180,E1 -4012.062,E2 -4012.062} C_VEL
LIN {X 0,Y 538.922,Z 226.869,A -85,B 0,C 180,E1 -4014.067,E2 -4014.067} C_VEL
LIN {X 0,Y 538.878,Z 234.02,A -85,B 0,C 180,E1 -4016.583,E2 -4016.583} C_VEL
LIN {X 0,Y 538.629,Z 242.498,A -85,B 0,C 180,E1 -4019.448,E2 -4019.448} C_VEL
LIN {X 0,Y 538.415,Z 250.234,A -85,B 0,C 180,E1 -4021.971,E2 -4021.971} C_VEL
LIN {X 0,Y 538.248,Z 259.48,A -85,B 0,C 180,E1 -4024.89,E2 -4024.89} C_VEL
LIN {X 0,Y 538.094,Z 269.686,A -85,B 0,C 180,E1 -4028.022,E2 -4028.022} C_VEL
LIN {X 0,Y 537.934,Z 279.393,A -85,B 0,C 180,E1 -4030.936,E2 -4030.936} C_VEL
LIN {X 0,Y 537.822,Z 290.26,A -85,B 0,C 180,E1 -4034.073,E2 -4034.073} C_VEL
LIN {X 0,Y 537.726,Z 299.469,A -85,B 0,C 180,E1 -4036.658,E2 -4036.658} C_VEL
LIN {X 0,Y 539.227,Z 309.867,A -85,B 0,C 180,E1 -4036.912,E2 -4036.912} C_VEL
LIN {X 0,Y 539.037,Z 322.048,A -85,B 0,C 180,E1 -4037.29,E2 -4037.29} C_VEL
LIN {X 0,Y 538.822,Z 333.132,A -85,B 0,C 180,E1 -4037.763,E2 -4037.763} C_VEL
LIN {X 0,Y 538.629,Z 344.163,A -85,B 0,C 180,E1 -4038.371,E2 -4038.371} C_VEL
LIN {X 0,Y 538.378,Z 355.745,A -85,B 0,C 180,E1 -4039.184,E2 -4039.184} C_VEL
LIN {X 0,Y 538.199,Z 365.516,A -85,B 0,C 180,E1 -4040.036,E2 -4040.036} C_VEL
LIN {X 0,Y 538.015,Z 374.405,A -85,B 0,C 180,E1 -4040.982,E2 -4040.982} C_VEL
LIN {X 0,Y 537.829,Z 383.004,A -85,B 0,C 180,E1 -4042.114,E2 -4042.114} C_VEL
LIN {X 0,Y 537.683,Z 390.75,A -85,B 0,C 180,E1 -4043.409,E2 -4043.409} C_VEL
LIN {X 0,Y 537.676,Z 395.366,A -85,B 0,C 180,E1 -4044.374,E2 -4044.374} C_VEL
LIN {X 0,Y 537.557,Z 399.677,A -85,B 0,C 180,E1 -4045.501,E2 -4045.501} C_VEL
LIN {X 0,Y 537.591,Z 401.958,A -85,B 0,C 180,E1 -4046.252,E2 -4046.252} C_VEL
LIN {X 0,Y 537.551,Z 403.807,A -85,B 0,C 180,E1 -4047.002,E2 -4047.002} C_VEL
LIN {X 0,Y 537.451,Z 406.182,A -85,B 0,C 180,E1 -4048.501,E2 -4048.501} C_VEL
LIN {X 0,Y 537.442,Z 407,A -85,B 0,C 180,E1 -4050,E2 -4050} C_VEL
LIN {X 0,Y 537.451,Z 406.183,A -85,B 0,C 180,E1 -4051.499,E2 -4051.499} C_VEL
LIN {X 0,Y 537.551,Z 403.81,A -85,B 0,C 180,E1 -4052.998,E2 -4052.998} C_VEL
LIN {X 0,Y 537.603,Z 400.895,A -85,B 0,C 180,E1 -4054.123,E2 -4054.123} C_VEL
LIN {X 0,Y 537.587,Z 396.947,A -85,B 0,C 180,E1 -4055.251,E2 -4055.251} C_VEL
LIN {X 0,Y 537.645,Z 392.123,A -85,B 0,C 180,E1 -4056.327,E2 -4056.327} C_VEL
LIN {X 0,Y 537.791,Z 385.465,A -85,B 0,C 180,E1 -4057.509,E2 -4057.509} C_VEL
LIN {X 0,Y 537.973,Z 377.475,A -85,B 0,C 180,E1 -4058.641,E2 -4058.641} C_VEL
LIN {X 0,Y 538.119,Z 369.284,A -85,B 0,C 180,E1 -4059.586,E2 -4059.586} C_VEL
LIN {X 0,Y 538.375,Z 359.232,A -85,B 0,C 180,E1 -4060.531,E2 -4060.531} C_VEL
LIN {X 0,Y 538.521,Z 349.299,A -85,B 0,C 180,E1 -4061.289,E2 -4061.289} C_VEL
LIN {X 0,Y 538.709,Z 338.234,A -85,B 0,C 180,E1 -4061.968,E2 -4061.968} C_VEL
LIN {X 0,Y 538.941,Z 325.539,A -85,B 0,C 180,E1 -4062.569,E2 -4062.569} C_VEL
LIN {X 0,Y 539.184,Z 312.379,A -85,B 0,C 180,E1 -4063.018,E2 -4063.018} C_VEL
LIN {X 0,Y 538.993,Z 307.269,A -85,B 0,C 180,E1 -4063.154,E2 -4063.154} C_VEL
LIN {X 0,Y 537.726,Z 299.042,A -85,B 0,C 180,E1 -4063.366,E2 -4063.366} C_VEL
LIN {X 0,Y 537.815,Z 288.52,A -85,B 0,C 180,E1 -4066.317,E2 -4066.317} C_VEL
LIN {X 0,Y 537.921,Z 278.781,A -85,B 0,C 180,E1 -4069.064,E2 -4069.064} C_VEL
LIN {X 0,Y 538.051,Z 267.829,A -85,B 0,C 180,E1 -4072.259,E2 -4072.259} C_VEL
LIN {X 0,Y 538.102,Z 258.314,A -85,B 0,C 180,E1 -4075.118,E2 -4075.118} C_VEL
LIN {X 0,Y 538.252,Z 249.068,A -85,B 0,C 180,E1 -4078.038,E2 -4078.038} C_VEL
LIN {X 0,Y 538.528,Z 240.254,A -85,B 0,C 180,E1 -4081.031,E2 -4081.031} C_VEL
LIN {X 0,Y 538.838,Z 233.842,A -85,B 0,C 180,E1 -4083.411,E2 -4083.411} C_VEL
LIN {X 0,Y 539.04,Z 228.941,A -85,B 0,C 180,E1 -4085.464,E2 -4085.464} C_VEL
LIN {X 0,Y 538.723,Z 225.24,A -85,B 0,C 180,E1 -4087.27,E2 -4087.27} C_VEL
LIN {X 0,Y 538.036,Z 221.469,A -85,B 0,C 180,E1 -4089.585,E2 -4089.585} C_VEL
LIN {X 0,Y 538.032,Z 221.469,A -85,B 0,C 180,E1 -4091.879,E2 -4091.879} C_VEL
LIN {X 0,Y 538.011,Z 221.47,A -85,B 0,C 180,E1 -4094.862,E2 -4094.862} C_VEL
LIN {X 0,Y 538.023,Z 221.469,A -85,B 0,C 180,E1 -4097.214,E2 -4097.214} C_VEL
LIN {X 0,Y 538.027,Z 221.469,A -85,B 0,C 180,E1 -4100.203,E2 -4100.203} C_VEL
LIN {X 0,Y 538.029,Z 221.47,A -85,B 0,C 180,E1 -4103.067,E2 -4103.067} C_VEL
LIN {X 0,Y 537.991,Z 221.475,A -85,B 0,C 180,E1 -4104.915,E2 -4104.915} C_VEL
LIN {X 0,Y 537.959,Z 223.793,A -85,B 0,C 180,E1 -4107.613,E2 -4107.613} C_VEL
LIN {X 0,Y 537.888,Z 226.279,A -85,B 0,C 180,E1 -4110.231,E2 -4110.231} C_VEL
LIN {X 0,Y 537.823,Z 228.782,A -85,B 0,C 180,E1 -4112.783,E2 -4112.783} C_VEL
LIN {X 0,Y 537.77,Z 231.282,A -85,B 0,C 180,E1 -4115.279,E2 -4115.279} C_VEL
LIN {X 0,Y 537.692,Z 234.619,A -85,B 0,C 180,E1 -4118.532,E2 -4118.532} C_VEL
LIN {X 0,Y 537.618,Z 237.153,A -85,B 0,C 180,E1 -4120.925,E2 -4120.925} C_VEL
LIN {X 0,Y 537.63,Z 239.615,A -85,B 0,C 180,E1 -4123.286,E2 -4123.286} C_VEL
LIN {X 0,Y 537.589,Z 242.15,A -85,B 0,C 180,E1 -4125.618,E2 -4125.618} C_VEL
LIN {X 0,Y 537.585,Z 244.555,A -85,B 0,C 180,E1 -4127.759,E2 -4127.759} C_VEL
LIN {X 0,Y 539.184,Z 254.479,A -85,B 0,C 180,E1 -4128.061,E2 -4128.061} C_VEL
LIN {X 0,Y 539.025,Z 267.427,A -85,B 0,C 180,E1 -4128.522,E2 -4128.522} C_VEL
LIN {X 0,Y 538.81,Z 279.301,A -85,B 0,C 180,E1 -4129.098,E2 -4129.098} C_VEL
LIN {X 0,Y 538.529,Z 289.918,A -85,B 0,C 180,E1 -4129.758,E2 -4129.758} C_VEL
LIN {X 0,Y 538.303,Z 300.755,A -85,B 0,C 180,E1 -4130.607,E2 -4130.607} C_VEL
LIN {X 0,Y 538.136,Z 310.455,A -85,B 0,C 180,E1 -4131.551,E2 -4131.551} C_VEL
LIN {X 0,Y 537.911,Z 318.404,A -85,B 0,C 180,E1 -4132.493,E2 -4132.493} C_VEL
LIN {X 0,Y 537.827,Z 325.694,A -85,B 0,C 180,E1 -4133.544,E2 -4133.544} C_VEL
LIN {X 0,Y 537.617,Z 332.405,A -85,B 0,C 180,E1 -4134.75,E2 -4134.75} C_VEL
LIN {X 0,Y 537.633,Z 337.337,A -85,B 0,C 180,E1 -4135.877,E2 -4135.877} C_VEL
LIN {X 0,Y 537.604,Z 341.159,A -85,B 0,C 180,E1 -4137.003,E2 -4137.003} C_VEL
LIN {X 0,Y 537.457,Z 344.695,A -85,B 0,C 180,E1 -4138.501,E2 -4138.501} C_VEL
LIN {X 0,Y 537.442,Z 345.864,A -85,B 0,C 180,E1 -4139.251,E2 -4139.251} C_VEL
LIN {X 0,Y 537.441,Z 346.943,A -85,B 0,C 180,E1 -4140.749,E2 -4140.749} C_VEL
LIN {X 0,Y 537.489,Z 346.489,A -85,B 0,C 180,E1 -4142.248,E2 -4142.248} C_VEL
LIN {X 0,Y 537.547,Z 345.635,A -85,B 0,C 180,E1 -4142.998,E2 -4142.998} C_VEL
LIN {X 0,Y 537.57,Z 344.382,A -85,B 0,C 180,E1 -4143.748,E2 -4143.748} C_VEL
LIN {X 0,Y 537.517,Z 341.752,A -85,B 0,C 180,E1 -4144.875,E2 -4144.875} C_VEL
LIN {X 0,Y 537.614,Z 338.115,A -85,B 0,C 180,E1 -4146.003,E2 -4146.003} C_VEL
LIN {X 0,Y 537.658,Z 333.366,A -85,B 0,C 180,E1 -4147.133,E2 -4147.133} C_VEL
LIN {X 0,Y 537.79,Z 327.353,A -85,B 0,C 180,E1 -4148.265,E2 -4148.265} C_VEL
LIN {X 0,Y 537.917,Z 319.86,A -85,B 0,C 180,E1 -4149.4,E2 -4149.4} C_VEL
LIN {X 0,Y 538.076,Z 312.184,A -85,B 0,C 180,E1 -4150.346,E2 -4150.346} C_VEL
LIN {X 0,Y 538.321,Z 302.802,A -85,B 0,C 180,E1 -4151.293,E2 -4151.293} C_VEL
LIN {X 0,Y 538.466,Z 292.359,A -85,B 0,C 180,E1 -4152.15,E2 -4152.15} C_VEL
LIN {X 0,Y 538.786,Z 280.737,A -85,B 0,C 180,E1 -4152.908,E2 -4152.908} C_VEL
LIN {X 0,Y 538.997,Z 268.338,A -85,B 0,C 180,E1 -4153.526,E2 -4153.526} C_VEL
LIN {X 0,Y 539.155,Z 255.268,A -85,B 0,C 180,E1 -4154.003,E2 -4154.003} C_VEL
LIN {X 0,Y 538.748,Z 250.805,A -85,B 0,C 180,E1 -4154.137,E2 -4154.137} C_VEL
LIN {X 0,Y 537.553,Z 244.191,A -85,B 0,C 180,E1 -4154.335,E2 -4154.335} C_VEL
LIN {X 0,Y 537.55,Z 240.42,A -85,B 0,C 180,E1 -4157.5,E2 -4157.5} C_VEL
LIN {X 0,Y 537.555,Z 237.686,A -85,B 0,C 180,E1 -4159.872,E2 -4159.872} C_VEL
LIN {X 0,Y 537.563,Z 234.947,A -85,B 0,C 180,E1 -4162.281,E2 -4162.281} C_VEL
LIN {X 0,Y 537.601,Z 232.125,A -85,B 0,C 180,E1 -4164.73,E2 -4164.73} C_VEL
LIN {X 0,Y 537.66,Z 229.191,A -85,B 0,C 180,E1 -4167.269,E2 -4167.269} C_VEL
LIN {X 0,Y 537.664,Z 225.666,A -85,B 0,C 180,E1 -4170.377,E2 -4170.377} C_VEL
LIN {X 0,Y 537.683,Z 222.328,A -85,B 0,C 180,E1 -4173.297,E2 -4173.297} C_VEL
LIN {X 0,Y 537.731,Z 221.507,A -85,B 0,C 180,E1 -4174.194,E2 -4174.194} C_VEL
LIN {X 0,Y 537.813,Z 221.497,A -85,B 0,C 180,E1 -4174.882,E2 -4174.882} C_VEL
LIN {X 0,Y 537.201,Z 221.574,A -85,B 0,C 180,E1 -4175.507,E2 -4175.507} C_VEL
LIN {X 0,Y 534.398,Z 221.92,A -85,B 0,C 180,E1 -4176.523,E2 -4176.523} C_VEL
LIN {X 0,Y 532.015,Z 222.213,A -85,B 0,C 180,E1 -4177.341,E2 -4177.341} C_VEL
LIN {X 0,Y 531.01,Z 222.343,A -85,B 0,C 180,E1 -4177.972,E2 -4177.972} C_VEL
LIN {X 0,Y 530.94,Z 222.347,A -85,B 0,C 180,E1 -4178.185,E2 -4178.185} C_VEL
LIN {X 0,Y 530.987,Z 222.34,A -85,B 0,C 180,E1 -4181.023,E2 -4181.023} C_VEL
LIN {X 0,Y 530.949,Z 222.351,A -85,B 0,C 180,E1 -4183.497,E2 -4183.497} C_VEL
LIN {X 0,Y 530.941,Z 222.346,A -85,B 0,C 180,E1 -4186.502,E2 -4186.502} C_VEL
LIN {X 0,Y 530.952,Z 222.347,A -85,B 0,C 180,E1 -4189.564,E2 -4189.564} C_VEL
LIN {X 0,Y 530.928,Z 222.351,A -85,B 0,C 180,E1 -4192.583,E2 -4192.583} C_VEL
LIN {X 0,Y 530.969,Z 222.342,A -85,B 0,C 180,E1 -4195.308,E2 -4195.308} C_VEL
LIN {X 0,Y 530.968,Z 222.345,A -85,B 0,C 180,E1 -4198.031,E2 -4198.031} C_VEL
LIN {X 0,Y 530.992,Z 222.34,A -85,B 0,C 180,E1 -4200.875,E2 -4200.875} C_VEL
LIN {X 0,Y 530.992,Z 222.34,A -85,B 0,C 180,E1 -4203.255,E2 -4203.255} C_VEL
LIN {X 0,Y 530.963,Z 222.348,A -85,B 0,C 180,E1 -4205.967,E2 -4205.967} C_VEL
LIN {X 0,Y 531.004,Z 222.341,A -85,B 0,C 180,E1 -4209.062,E2 -4209.062} C_VEL
LIN {X 0,Y 530.988,Z 222.345,A -85,B 0,C 180,E1 -4211.478,E2 -4211.478} C_VEL
LIN {X 0,Y 530.997,Z 222.343,A -85,B 0,C 180,E1 -4214.65,E2 -4214.65} C_VEL
LIN {X 0,Y 531.027,Z 222.335,A -85,B 0,C 180,E1 -4217.775,E2 -4217.775} C_VEL
LIN {X 0,Y 530.977,Z 222.344,A -85,B 0,C 180,E1 -4220.092,E2 -4220.092} C_VEL
LIN {X 0,Y 531.013,Z 222.336,A -85,B 0,C 180,E1 -4223.159,E2 -4223.159} C_VEL
LIN {X 0,Y 530.978,Z 222.342,A -85,B 0,C 180,E1 -4225.445,E2 -4225.445} C_VEL
LIN {X 0,Y 531.136,Z 222.327,A -85,B 0,C 180,E1 -4227.725,E2 -4227.725} C_VEL
LIN {X 0,Y 531.135,Z 222.324,A -85,B 0,C 180,E1 -4230,E2 -4230} C_VEL
LIN {X 0,Y 531.101,Z 222.328,A -85,B 0,C 180,E1 -4233.034,E2 -4233.034} C_VEL
LIN {X 0,Y 530.788,Z 222.393,A -85,B 0,C 180,E1 -4235.699,E2 -4235.699} C_VEL
LIN {X 0,Y 530.8,Z 226.775,A -85,B 0,C 180,E1 -4237.608,E2 -4237.608} C_VEL
LIN {X 0,Y 530.757,Z 233.73,A -85,B 0,C 180,E1 -4240.683,E2 -4240.683} C_VEL
LIN {X 0,Y 530.687,Z 240.707,A -85,B 0,C 180,E1 -4243.791,E2 -4243.791} C_VEL
LIN {X 0,Y 530.67,Z 245.906,A -85,B 0,C 180,E1 -4246.148,E2 -4246.148} C_VEL
LIN {X 0,Y 530.636,Z 251.126,A -85,B 0,C 180,E1 -4248.534,E2 -4248.534} C_VEL
LIN {X 0,Y 530.566,Z 258.202,A -85,B 0,C 180,E1 -4251.771,E2 -4251.771} C_VEL
LIN {X 0,Y 530.504,Z 263.582,A -85,B 0,C 180,E1 -4254.248,E2 -4254.248} C_VEL
LIN {X 0,Y 530.496,Z 268.132,A -85,B 0,C 180,E1 -4256.4,E2 -4256.4} C_VEL
LIN {X 0,Y 531.619,Z 276.482,A -85,B 0,C 180,E1 -4256.671,E2 -4256.671} C_VEL
LIN {X 0,Y 531.435,Z 288.412,A -85,B 0,C 180,E1 -4257.145,E2 -4257.145} C_VEL
LIN {X 0,Y 531.265,Z 297.933,A -85,B 0,C 180,E1 -4257.677,E2 -4257.677} C_VEL
LIN {X 0,Y 531.104,Z 307.179,A -85,B 0,C 180,E1 -4258.342,E2 -4258.342} C_VEL
LIN {X 0,Y 531.011,Z 314.478,A -85,B 0,C 180,E1 -4258.989,E2 -4258.989} C_VEL
LIN {X 0,Y 530.84,Z 321.666,A -85,B 0,C 180,E1 -4259.767,E2 -4259.767} C_VEL
LIN {X 0,Y 530.701,Z 327.913,A -85,B 0,C 180,E1 -4260.594,E2 -4260.594} C_VEL
LIN {X 0,Y 530.631,Z 333.696,A -85,B 0,C 180,E1 -4261.545,E2 -4261.545} C_VEL
LIN {X 0,Y 530.517,Z 338.083,A -85,B 0,C 180,E1 -4262.447,E2 -4262.447} C_VEL
LIN {X 0,Y 530.484,Z 341.764,A -85,B 0,C 180,E1 -4263.421,E2 -4263.421} C_VEL
LIN {X 0,Y 530.457,Z 344.197,A -85,B 0,C 180,E1 -4264.269,E2 -4264.269} C_VEL
LIN {X 0,Y 530.426,Z 345.313,A -85,B 0,C 180,E1 -4264.766,E2 -4264.766} C_VEL
LIN {X 0,Y 530.4,Z 347.182,A -85,B 0,C 180,E1 -4266.072,E2 -4266.072} C_VEL
LIN {X 0,Y 530.337,Z 347.402,A -85,B 0,C 180,E1 -4267.56,E2 -4267.56} C_VEL
LIN {X 0,Y 530.355,Z 346.528,A -85,B 0,C 180,E1 -4268.57,E2 -4268.57} C_VEL
LIN {X 0,Y 530.444,Z 344.295,A -85,B 0,C 180,E1 -4269.784,E2 -4269.784} C_VEL
LIN {X 0,Y 530.511,Z 340.83,A -85,B 0,C 180,E1 -4270.964,E2 -4270.964} C_VEL
LIN {X 0,Y 530.591,Z 335.186,A -85,B 0,C 180,E1 -4272.274,E2 -4272.274} C_VEL
LIN {X 0,Y 530.669,Z 329.599,A -85,B 0,C 180,E1 -4273.247,E2 -4273.247} C_VEL
LIN {X 0,Y 530.819,Z 322.714,A -85,B 0,C 180,E1 -4274.199,E2 -4274.199} C_VEL
LIN {X 0,Y 530.934,Z 315.987,A -85,B 0,C 180,E1 -4274.953,E2 -4274.953} C_VEL
LIN {X 0,Y 531.084,Z 308.881,A -85,B 0,C 180,E1 -4275.61,E2 -4275.61} C_VEL
LIN {X 0,Y 531.216,Z 302.007,A -85,B 0,C 180,E1 -4276.14,E2 -4276.14} C_VEL
LIN {X 0,Y 531.354,Z 293.512,A -85,B 0,C 180,E1 -4276.674,E2 -4276.674} C_VEL
LIN {X 0,Y 531.498,Z 284.477,A -85,B 0,C 180,E1 -4277.119,E2 -4277.119} C_VEL
LIN {X 0,Y 531.513,Z 275.058,A -85,B 0,C 180,E1 -4277.467,E2 -4277.467} C_VEL
LIN {X 0,Y 530.511,Z 268.257,A -85,B 0,C 180,E1 -4277.684,E2 -4277.684} C_VEL
LIN {X 0,Y 530.553,Z 262.241,A -85,B 0,C 180,E1 -4280.518,E2 -4280.518} C_VEL
LIN {X 0,Y 530.559,Z 255.866,A -85,B 0,C 180,E1 -4283.409,E2 -4283.409} C_VEL
LIN {X 0,Y 530.666,Z 248.895,A -85,B 0,C 180,E1 -4286.549,E2 -4286.549} C_VEL
LIN {X 0,Y 530.64,Z 242.555,A -85,B 0,C 180,E1 -4289.416,E2 -4289.416} C_VEL
LIN {X 0,Y 530.658,Z 235.75,A -85,B 0,C 180,E1 -4292.384,E2 -4292.384} C_VEL
LIN {X 0,Y 530.694,Z 229.807,A -85,B 0,C 180,E1 -4294.927,E2 -4294.927} C_VEL
LIN {X 0,Y 530.781,Z 222.375,A -85,B 0,C 180,E1 -4298.042,E2 -4298.042} C_VEL
LIN {X 0,Y 531.02,Z 222.343,A -85,B 0,C 180,E1 -4299.998,E2 -4299.998} C_VEL
LIN {X 0,Y 530.973,Z 222.347,A -85,B 0,C 180,E1 -4303.07,E2 -4303.07} C_VEL
LIN {X 0,Y 531.02,Z 222.34,A -85,B 0,C 180,E1 -4305.436,E2 -4305.436} C_VEL
LIN {X 0,Y 531.039,Z 222.339,A -85,B 0,C 180,E1 -4308.55,E2 -4308.55} C_VEL
LIN {X 0,Y 531.058,Z 222.337,A -85,B 0,C 180,E1 -4311.629,E2 -4311.629} C_VEL
LIN {X 0,Y 531.115,Z 222.328,A -85,B 0,C 180,E1 -4314.685,E2 -4314.685} C_VEL
LIN {X 0,Y 531.143,Z 222.327,A -85,B 0,C 180,E1 -4317.725,E2 -4317.725} C_VEL
LIN {X 0,Y 531.154,Z 222.323,A -85,B 0,C 180,E1 -4320.758,E2 -4320.758} C_VEL
LIN {X 0,Y 531.106,Z 222.329,A -85,B 0,C 180,E1 -4323.034,E2 -4323.034} C_VEL
LIN {X 0,Y 531.071,Z 222.336,A -85,B 0,C 180,E1 -4326.077,E2 -4326.077} C_VEL
LIN {X 0,Y 531.057,Z 222.338,A -85,B 0,C 180,E1 -4328.37,E2 -4328.37} C_VEL
LIN {X 0,Y 531.055,Z 222.336,A -85,B 0,C 180,E1 -4331.672,E2 -4331.672} C_VEL
LIN {X 0,Y 531.035,Z 222.338,A -85,B 0,C 180,E1 -4334.956,E2 -4334.956} C_VEL
LIN {X 0,Y 530.984,Z 222.346,A -85,B 0,C 180,E1 -4337.723,E2 -4337.723} C_VEL
LIN {X 0,Y 531.028,Z 222.34,A -85,B 0,C 180,E1 -4340.127,E2 -4340.127} C_VEL
LIN {X 0,Y 530.948,Z 222.351,A -85,B 0,C 180,E1 -4342.573,E2 -4342.573} C_VEL
LIN {X 0,Y 530.972,Z 222.348,A -85,B 0,C 180,E1 -4345.059,E2 -4345.059} C_VEL
LIN {X 0,Y 531.014,Z 222.343,A -85,B 0,C 180,E1 -4347.596,E2 -4347.596} C_VEL
LIN {X 0,Y 530.969,Z 222.346,A -85,B 0,C 180,E1 -4350.644,E2 -4350.644} C_VEL
LIN {X 0,Y 530.965,Z 222.349,A -85,B 0,C 180,E1 -4353.5,E2 -4353.5} C_VEL
LIN {X 0,Y 530.948,Z 222.349,A -85,B 0,C 180,E1 -4356.153,E2 -4356.153} C_VEL
LIN {X 0,Y 530.969,Z 222.346,A -85,B 0,C 180,E1 -4358.654,E2 -4358.654} C_VEL
LIN {X 0,Y 530.995,Z 222.344,A -85,B 0,C 180,E1 -4361.436,E2 -4361.436} C_VEL
LIN {X 0,Y 530.977,Z 222.346,A -85,B 0,C 180,E1 -4364.548,E2 -4364.548} C_VEL
LIN {X 0,Y 530.984,Z 222.346,A -85,B 0,C 180,E1 -4367.834,E2 -4367.834} C_VEL
LIN {X 0,Y 530.991,Z 222.344,A -85,B 0,C 180,E1 -4370.557,E2 -4370.557} C_VEL
LIN {X 0,Y 531.013,Z 222.49,A -85,B 0,C 180,E1 -4371.836,E2 -4371.836} C_VEL
LIN {X 0,Y 531.971,Z 228.385,A -85,B 0,C 180,E1 -4374.093,E2 -4374.093} C_VEL
LIN {X 0,Y 531.921,Z 234.674,A -85,B 0,C 180,E1 -4376.345,E2 -4376.345} C_VEL
LIN {X 0,Y 531.67,Z 243.087,A -85,B 0,C 180,E1 -4379.229,E2 -4379.229} C_VEL
LIN {X 0,Y 531.399,Z 251.446,A -85,B 0,C 180,E1 -4381.998,E2 -4381.998} C_VEL
LIN {X 0,Y 531.21,Z 260.661,A -85,B 0,C 180,E1 -4384.953,E2 -4384.953} C_VEL
LIN {X 0,Y 531.048,Z 270.04,A -85,B 0,C 180,E1 -4387.88,E2 -4387.88} C_VEL
LIN {X 0,Y 530.91,Z 279.221,A -85,B 0,C 180,E1 -4390.674,E2 -4390.674} C_VEL
LIN {X 0,Y 530.75,Z 290.003,A -85,B 0,C 180,E1 -4393.855,E2 -4393.855} C_VEL
LIN {X 0,Y 530.655,Z 299.004,A -85,B 0,C 180,E1 -4396.477,E2 -4396.477} C_VEL
LIN {X 0,Y 532.276,Z 311.168,A -85,B 0,C 180,E1 -4396.786,E2 -4396.786} C_VEL
LIN {X 0,Y 532.048,Z 324.047,A -85,B 0,C 180,E1 -4397.217,E2 -4397.217} C_VEL
LIN {X 0,Y 531.788,Z 336.334,A -85,B 0,C 180,E1 -4397.793,E2 -4397.793} C_VEL
LIN {X 0,Y 531.546,Z 347.208,A -85,B 0,C 180,E1 -4398.449,E2 -4398.449} C_VEL
LIN {X 0,Y 531.347,Z 358.786,A -85,B 0,C 180,E1 -4399.329,E2 -4399.329} C_VEL
LIN {X 0,Y 531.069,Z 368.827,A -85,B 0,C 180,E1 -4400.286,E2 -4400.286} C_VEL
LIN {X 0,Y 530.853,Z 378.565,A -85,B 0,C 180,E1 -4401.435,E2 -4401.435} C_VEL
LIN {X 0,Y 530.681,Z 386.322,A -85,B 0,C 180,E1 -4402.581,E2 -4402.581} C_VEL
LIN {X 0,Y 530.585,Z 393.468,A -85,B 0,C 180,E1 -4403.917,E2 -4403.917} C_VEL
LIN {X 0,Y 530.459,Z 398.217,A -85,B 0,C 180,E1 -4405.06,E2 -4405.06} C_VEL
LIN {X 0,Y 530.516,Z 401.854,A -85,B 0,C 180,E1 -4406.202,E2 -4406.202} C_VEL
LIN {X 0,Y 530.457,Z 403.724,A -85,B 0,C 180,E1 -4406.962,E2 -4406.962} C_VEL
LIN {X 0,Y 530.411,Z 405.126,A -85,B 0,C 180,E1 -4407.722,E2 -4407.722} C_VEL
LIN {X 0,Y 530.344,Z 406.736,A -85,B 0,C 180,E1 -4409.241,E2 -4409.241} C_VEL
LIN {X 0,Y 530.343,Z 406.953,A -85,B 0,C 180,E1 -4410,E2 -4410} C_VEL
LIN {X 0,Y 530.361,Z 406.126,A -85,B 0,C 180,E1 -4411.519,E2 -4411.519} C_VEL
LIN {X 0,Y 530.411,Z 405.127,A -85,B 0,C 180,E1 -4412.278,E2 -4412.278} C_VEL
LIN {X 0,Y 530.457,Z 403.724,A -85,B 0,C 180,E1 -4413.038,E2 -4413.038} C_VEL
LIN {X 0,Y 530.522,Z 400.77,A -85,B 0,C 180,E1 -4414.178,E2 -4414.178} C_VEL
LIN {X 0,Y 530.524,Z 396.762,A -85,B 0,C 180,E1 -4415.321,E2 -4415.321} C_VEL
LIN {X 0,Y 530.596,Z 391.002,A -85,B 0,C 180,E1 -4416.579,E2 -4416.579} C_VEL
LIN {X 0,Y 530.728,Z 383.852,A -85,B 0,C 180,E1 -4417.801,E2 -4417.801} C_VEL
LIN {X 0,Y 530.909,Z 375.479,A -85,B 0,C 180,E1 -4418.948,E2 -4418.948} C_VEL
LIN {X 0,Y 531.081,Z 366.882,A -85,B 0,C 180,E1 -4419.906,E2 -4419.906} C_VEL
LIN {X 0,Y 531.334,Z 356.267,A -85,B 0,C 180,E1 -4420.865,E2 -4420.865} C_VEL
LIN {X 0,Y 531.556,Z 344.427,A -85,B 0,C 180,E1 -4421.722,E2 -4421.722} C_VEL
LIN {X 0,Y 531.823,Z 332.28,A -85,B 0,C 180,E1 -4422.401,E2 -4422.401} C_VEL
